    !************************************************
    ! Function    :     User interface message
    ! Programmer  :     Philippe Fleischmann
    ! Date        :     2019.02.22
    !***************** ETH Zurich *******************
    !
    FUNC string f_RRC_UIMsg(string stMsgHeader,string stMsgL1,\string stMsgL2,\string stMsgL3,\string stMsgL4,\string stMsgL5,string stBtn1\string stBtn2\string stBtn3\string stBtn4\string stBtn5,icondata icIcon)
        VAR num nAnswer;
        VAR string stMsg{5};
        VAR string stBtn{5};
        VAR string stAnswer;
        !
        ! Initialize variables
        stMsg:=["","","","",""];
        stBtn:=["","","","",""];
        !
        ! Load meassge
        stMsg{1}:=stMsgL1;
        IF Present(stMsgL2) stMsg{2}:=stMsgL2;
        IF Present(stMsgL3) stMsg{3}:=stMsgL3;
        IF Present(stMsgL4) stMsg{4}:=stMsgL4;
        IF Present(stMsgL5) stMsg{5}:=stMsgL5;
        !
        ! Load buttons
        stBtn{1}:=stBtn1;
        IF Present(stBtn2) stBtn{2}:=stBtn2;
        IF Present(stBtn3) stBtn{3}:=stBtn3;
        IF Present(stBtn4) stBtn{4}:=stBtn4;
        IF Present(stBtn5) stBtn{5}:=stBtn5;
        !
        ! Msg for user
        nAnswer:=UIMessageBox(
            \Header:=stMsgHeader
            \MsgArray:=stMsg
            \BtnArray:=stBtn
            \Icon:=icIcon);
        !
        ! handle user answer
        IF nAnswer=1 stAnswer:=stBtn{1};
        IF nAnswer=2 stAnswer:=stBtn{2};
        IF nAnswer=3 stAnswer:=stBtn{3};
        IF nAnswer=4 stAnswer:=stBtn{4};
        IF nAnswer=5 stAnswer:=stBtn{5};
        !
        ! Return user answer as string
        RETURN stAnswer;
    ERROR
        ! Placeholder for Error Code...
    ENDFUNC

    !************************************************
    ! Function    :     User interface numerical entry
    ! Programmer  :     Philippe Fleischmann
    ! Date        :     2019.02.22
    !***************** ETH Zurich *******************
    !
    FUNC num f_RRC_UINumEntry(string stMsgHeader,string stMsgL1,\string stMsgL2,\string stMsgL3,\string stMsgL4,\string stMsgL5,num nMin,num nMax,\num nDefault,icondata icIcon)
        VAR string stMsg{5};
        VAR num nAnswer;
        VAR num nInitValue;
        !
        ! Initialize variables
        stMsg:=["","","","",""];
        nInitValue:=nMin;
        !
        ! Load meassge
        stMsg{1}:=stMsgL1;
        IF Present(stMsgL2) stMsg{2}:=stMsgL2;
        IF Present(stMsgL3) stMsg{3}:=stMsgL3;
        IF Present(stMsgL4) stMsg{4}:=stMsgL4;
        IF Present(stMsgL5) stMsg{5}:=stMsgL5;
        !
        ! Use default value when present
        IF Present(nDefault) nInitValue:=nDefault;
        !
        ! Msg for user
        nAnswer:=Round(UINumEntry(
            \Header:=stMsgHeader
            \MsgArray:=stMsg
            \Icon:=icIcon
            \InitValue:=nInitValue
            \MinValue:=nMin
            \MaxValue:=nMax)\Dec:=1);
        !
        ! Return user answer as string
        RETURN nAnswer;
    ERROR
        ! Placeholder for Error Code...
    ENDFUNC


ENDMODULE

--- Backups/vIRB4600-40-2.55-RW11/RAPID/TASK2/SYSMOD/RRC_Base_Feedback_Ctrl.sys ---
MODULE RRC_Base_Feedback_Ctrl(SYSMODULE)
    !***********************************************************************************
    !
    ! ETH Zurich / Robotic Fabrication Lab
    ! HIB C 13 / Stefano-Franscini-Platz 1
    ! CH-8093 Zurich
    !
    !***********************************************************************************
    !
    ! PROJECT     :  RRC - Rapid Robot Communication
    !
    ! FUNCTION    :  Base Feedback Library
    !
    ! AUTHOR      :  Philippe Fleischmann
    !
    ! EMAIL       :  rrc@arch.ethz.ch
    !
    ! HISTORY     :  2019.02.22
    !
    ! Copyright   :  ETH Zurich (CH) 2019
    !                - Philippe Fleischmann
    !                - Michael Lyrenmann
    !                - Gonzalo Casas
    !
    ! License     :  This code base is governed by an EULA (End-User License Agreement)
    !                which you have received together with the software.
    !                You are not allowed to use the software on a real robots
    !                without a signed EULA.
    !
    !                A copy of the EULA content is in the controller task (T_CTRL).
    !
    !***********************************************************************************

    !************************************************
    ! Function    :     Feedback add string
    ! Programmer  :     Philippe Fleischmann
    ! Date        :     2019.02.22
    !***************** ETH Zurich *******************
    !
    PROC r_RRC_FAddString(string stString)
        !
        ! Increase feedback string counter
        Incr n_RRC_CounterFStr{n_RRC_ChaNr};
        !
        ! Select string to add
        TEST n_RRC_CounterFStr{n_RRC_ChaNr}
        CASE 1:
            !
            ! Add string
            bm_RRC_ActSenMsgCtrl{n_RRC_ChaNr}.Data.St1:=stString;
        CASE 2:
            !
            ! Add string
            bm_RRC_ActSenMsgCtrl{n_RRC_ChaNr}.Data.St2:=stString;
        CASE 3:
            !
            ! Add string
            bm_RRC_ActSenMsgCtrl{n_RRC_ChaNr}.Data.St3:=stString;
        CASE 4:
            !
            ! Add string
            bm_RRC_ActSenMsgCtrl{n_RRC_ChaNr}.Data.St4:=stString;
        CASE 5:
            !
            ! Add string
            bm_RRC_ActSenMsgCtrl{n_RRC_ChaNr}.Data.St5:=stString;
        DEFAULT:
            !
            ! Program error
            r_RRC_ProgError;
        ENDTEST
        !
        ! Update string counter
        bm_RRC_ActSenMsgCtrl{n_RRC_ChaNr}.Data.St_Cnt:=n_RRC_CounterFStr{n_RRC_ChaNr};
        RETURN ;
    ERROR
        ! Placeholder for Error Code...
    ENDPROC

    !************************************************
    ! Function    :     Feedback add value
    ! Programmer  :     Philippe Fleischmann
    ! Date        :     2019.02.22
    !***************** ETH Zurich *******************
    !
    PROC r_RRC_FAddValue(num nValue)
        !
        ! Increase feedback value counter
        Incr n_RRC_CounterFVal{n_RRC_ChaNr};
        !
        ! Select value to add
        TEST n_RRC_CounterFVal{n_RRC_ChaNr}
        CASE 1:
            !
            ! Add value
            bm_RRC_ActSenMsgCtrl{n_RRC_ChaNr}.Data.V1:=nValue;
        CASE 2:
            !
            ! Add value
            bm_RRC_ActSenMsgCtrl{n_RRC_ChaNr}.Data.V2:=nValue;
        CASE 3:
            !
            ! Add value
            bm_RRC_ActSenMsgCtrl{n_RRC_ChaNr}.Data.V3:=nValue;
        CASE 4:
            !
            ! Add value
            bm_RRC_ActSenMsgCtrl{n_RRC_ChaNr}.Data.V4:=nValue;
        CASE 5:
            !
            ! Add value
            bm_RRC_ActSenMsgCtrl{n_RRC_ChaNr}.Data.V5:=nValue;
        CASE 6:
            !
            ! Add value
            bm_RRC_ActSenMsgCtrl{n_RRC_ChaNr}.Data.V6:=nValue;
        CASE 7:
            !
            ! Add value
            bm_RRC_ActSenMsgCtrl{n_RRC_ChaNr}.Data.V7:=nValue;
        CASE 8:
            !
            ! Add value
            bm_RRC_ActSenMsgCtrl{n_RRC_ChaNr}.Data.V8:=nValue;
        CASE 9:
            !
            ! Add value
            bm_RRC_ActSenMsgCtrl{n_RRC_ChaNr}.Data.V9:=nValue;
        CASE 10:
            !
            ! Add value
            bm_RRC_ActSenMsgCtrl{n_RRC_ChaNr}.Data.V10:=nValue;
        CASE 11:
            !
            ! Add value
            bm_RRC_ActSenMsgCtrl{n_RRC_ChaNr}.Data.V11:=nValue;
        CASE 12:
            !
            ! Add value
            bm_RRC_ActSenMsgCtrl{n_RRC_ChaNr}.Data.V12:=nValue;
        CASE 13:
            !
            ! Add value
            bm_RRC_ActSenMsgCtrl{n_RRC_ChaNr}.Data.V13:=nValue;
        CASE 14:
            !
            ! Add value
            bm_RRC_ActSenMsgCtrl{n_RRC_ChaNr}.Data.V14:=nValue;
        CASE 15:
            !
            ! Add value
            bm_RRC_ActSenMsgCtrl{n_RRC_ChaNr}.Data.V15:=nValue;
        CASE 16:
            !
            ! Add value
            bm_RRC_ActSenMsgCtrl{n_RRC_ChaNr}.Data.V16:=nValue;
        CASE 17:
            !
            ! Add value
            bm_RRC_ActSenMsgCtrl{n_RRC_ChaNr}.Data.V17:=nValue;
        CASE 18:
            !
            ! Add value
            bm_RRC_ActSenMsgCtrl{n_RRC_ChaNr}.Data.V18:=nValue;
        CASE 19:
            !
            ! Add value
            bm_RRC_ActSenMsgCtrl{n_RRC_ChaNr}.Data.V19:=nValue;
        CASE 20:
            !
            ! Add value
            bm_RRC_ActSenMsgCtrl{n_RRC_ChaNr}.Data.V20:=nValue;
        CASE 21:
            !
            ! Add value
            bm_RRC_ActSenMsgCtrl{n_RRC_ChaNr}.Data.V21:=nValue;
        CASE 22:
            !
            ! Add value
            bm_RRC_ActSenMsgCtrl{n_RRC_ChaNr}.Data.V22:=nValue;
        CASE 23:
            !
            ! Add value
            bm_RRC_ActSenMsgCtrl{n_RRC_ChaNr}.Data.V23:=nValue;
        CASE 24:
            !
            ! Add value
            bm_RRC_ActSenMsgCtrl{n_RRC_ChaNr}.Data.V24:=nValue;
        CASE 25:
            !
            ! Add value
            bm_RRC_ActSenMsgCtrl{n_RRC_ChaNr}.Data.V25:=nValue;
        CASE 26:
            !
            ! Add value
            bm_RRC_ActSenMsgCtrl{n_RRC_ChaNr}.Data.V26:=nValue;
        CASE 27:
            !
            ! Add value
            bm_RRC_ActSenMsgCtrl{n_RRC_ChaNr}.Data.V27:=nValue;
        CASE 28:
            !
            ! Add value
            bm_RRC_ActSenMsgCtrl{n_RRC_ChaNr}.Data.V28:=nValue;
        CASE 29:
            !
            ! Add value
            bm_RRC_ActSenMsgCtrl{n_RRC_ChaNr}.Data.V29:=nValue;
        CASE 30:
            !
            ! Add value
            bm_RRC_ActSenMsgCtrl{n_RRC_ChaNr}.Data.V30:=nValue;
        DEFAULT:
            !
            ! Program error
            r_RRC_ProgError;
        ENDTEST
        !
        ! Update value counter
        bm_RRC_ActSenMsgCtrl{n_RRC_ChaNr}.Data.V_Cnt:=n_RRC_CounterFVal{n_RRC_ChaNr};
        RETURN ;
    ERROR
        ! Placeholder for Error Code...
    ENDPROC

    !************************************************
    ! Function    :     Feedback done
    ! Programmer  :     Philippe Fleischmann
    ! Date        :     2019.02.22
    !***************** ETH Zurich *******************
    !
    PROC r_RRC_FDone()
        !
        ! Add Sqz_ID from Client in Feedback ID
        bm_RRC_ActSenMsgCtrl{n_RRC_ChaNr}.Data.F_ID:=bm_RRC_RecBufferCtrl{n_RRC_ChaNr,n_RRC_ReadPtrRecBuf{n_RRC_ChaNr}}.Data.S_ID;
        !
        ! Instruction
        bm_RRC_ActSenMsgCtrl{n_RRC_ChaNr}.Data.Instr:=bm_RRC_RecBufferCtrl{n_RRC_ChaNr,n_RRC_ReadPtrRecBuf{n_RRC_ChaNr}}.Data.Instr;
        !
        ! Feedback
        bm_RRC_ActSenMsgCtrl{n_RRC_ChaNr}.Data.Feedb:="Controller Done";
        RETURN ;
    ERROR
        ! Placeholder for Error Code...
    ENDPROC

    !************************************************
    ! Function    :     Cycle Feedback done
    ! Programmer  :     Philippe Fleischmann
    ! Date        :     2019.02.22
    !***************** ETH Zurich *******************
    !
    PROC r_RRC_CyFDone()
        !
        ! Add cyclic jop Sqz_ID from cyclic job start instruction
        bm_RRC_ActSenMsgCtrl{n_RRC_ChaNr}.Data.F_ID:=n_RRC_CyJobStart_S_ID{n_RRC_ChaNr};
        !
        ! Add cyclic jop instruction
        bm_RRC_ActSenMsgCtrl{n_RRC_ChaNr}.Data.Instr:=st_RRC_CyclicJob{n_RRC_ChaNr};
        !
        ! Feedback
        bm_RRC_ActSenMsgCtrl{n_RRC_ChaNr}.Data.Feedb:="Controller Done";
        RETURN ;
    ERROR
        ! Placeholder for Error Code...
    ENDPROC

    !************************************************
    ! Function    :     Feedback error
    ! Programmer  :     Philippe Fleischmann
    ! Date        :     2019.02.22
    !***************** ETH Zurich *******************
    !
    PROC r_RRC_FError()
        !
        ! Feedback error with feedback code
        bm_RRC_ActSenMsgCtrl{n_RRC_ChaNr}.Data.Feedb:="Controller Done FError "+NumToStr(bm_RRC_RecBufferCtrl{n_RRC_ChaNr,n_RRC_ReadPtrRecBuf{n_RRC_ChaNr}}.Data.F_Lev,0);
        RETURN ;
    ERROR
        ! Placeholder for Error Code...
    ENDPROC
ENDMODULE

--- Backups/vIRB4600-40-2.55-RW11/RAPID/TASK2/SYSMOD/RRC_Base_Instructions_Ctrl.sys ---
MODULE RRC_Base_Instructions_Ctrl(SYSMODULE)
    !***********************************************************************************
    !
    ! ETH Zurich / Robotic Fabrication Lab
    ! HIB C 13 / Stefano-Franscini-Platz 1
    ! CH-8093 Zurich
    !
    !***********************************************************************************
    !
    ! PROJECT     :  RRC - Rapid Robot Communication
    !
    ! FUNCTION    :  Base Instracion Library for controller
    !
    ! AUTHOR      :  Philippe Fleischmann
    !
    ! EMAIL       :  rrc@arch.ethz.ch
    !
    ! HISTORY     :  2019.02.22
    !
    ! Copyright   :  ETH Zurich (CH) 2019
    !                - Philippe Fleischmann
    !                - Michael Lyrenmann
    !                - Gonzalo Casas
    !
    ! License     :  This code base is governed by an EULA (End-User License Agreement)
    !                which you have received together with the software.
    !                You are not allowed to use the software on a real robots
    !                without a signed EULA.
    !
    !                A copy of the EULA content is in the controller task (T_CTRL).
    !
    !***********************************************************************************

    !************************************************
    ! Function    :     Dummy
    ! Programmer  :     Philippe Fleischmann
    ! Date        :     2019.02.22
    !***************** ETH Zurich *******************
    !
    PROC r_RRC_Dummy()
        !
        ! Just a dummy procedure for communication tests
        !
        ! Read the current Sequnce ID
        n_RRC_Act_S_ID:=bm_RRC_RecBufferCtrl{n_RRC_ChaNr,n_RRC_ReadPtrRecBuf{n_RRC_ChaNr}}.Data.S_ID;
        !
        ! Feedback
        IF bm_RRC_RecBufferCtrl{n_RRC_ChaNr,n_RRC_ReadPtrRecBuf{n_RRC_ChaNr}}.Data.F_Lev>0 THEN
            !
            ! Cenerate feedback
            TEST bm_RRC_RecBufferCtrl{n_RRC_ChaNr,n_RRC_ReadPtrRecBuf{n_RRC_ChaNr}}.Data.F_Lev
            CASE 1:
                !nChaNr
                ! Instruction done
                r_RRC_FDone;
            DEFAULT:
                !
                ! Feedback not supported
                r_RRC_FError;
            ENDTEST
            !
            ! Move message in send buffer
            r_RRC_MovMsgToSenBufCtrl n_RRC_ChaNr;
        ENDIF
        RETURN ;
    ERROR
        ! Placeholder for Error Code...
    ENDPROC

    !************************************************
    ! Function    :     Read actual jointtarget
    ! Programmer  :     Philippe Fleischmann
    ! Date        :     2019.02.22
    !***************** ETH Zurich *******************
    !
    PROC r_RRC_GetJointT()
        !
        ! Read current joint position
        jp_RRC_Act:=CJointT(\TaskName:=st_RRC_ChaTask);
        !
        ! Add robot axis values to feedback
        r_RRC_FAddValue jp_RRC_Act.robax.rax_1;
        r_RRC_FAddValue jp_RRC_Act.robax.rax_2;
        r_RRC_FAddValue jp_RRC_Act.robax.rax_3;
        r_RRC_FAddValue jp_RRC_Act.robax.rax_4;
        r_RRC_FAddValue jp_RRC_Act.robax.rax_5;
        r_RRC_FAddValue jp_RRC_Act.robax.rax_6;
        !
        ! Add external axis values to feedback
        r_RRC_FAddValue jp_RRC_Act.extax.eax_a;
        r_RRC_FAddValue jp_RRC_Act.extax.eax_b;
        r_RRC_FAddValue jp_RRC_Act.extax.eax_c;
        r_RRC_FAddValue jp_RRC_Act.extax.eax_d;
        r_RRC_FAddValue jp_RRC_Act.extax.eax_e;
        r_RRC_FAddValue jp_RRC_Act.extax.eax_f;
        !
        ! Add cyclic feedback instruction done
        r_RRC_CyFDone;
        !
        ! Feedback
        IF bm_RRC_RecBufferCtrl{n_RRC_ChaNr,n_RRC_ReadPtrRecBuf{n_RRC_ChaNr}}.Data.F_Lev>1 THEN
            !
            ! Check additional feedback
            TEST bm_RRC_RecBufferCtrl{n_RRC_ChaNr,n_RRC_ReadPtrRecBuf{n_RRC_ChaNr}}.Data.F_Lev
            CASE 10001:
                !
                ! add robot position
                !* r_RRC_FPos bm_RRC_RecBufferRob{n_RRC_ChaNr,n_RRC_ReadPtrRecBuf}.Data.F_Lev;
            DEFAULT:
                !
                ! Not defined
                !
                ! Feedback not supported
                r_RRC_FError;
            ENDTEST
        ENDIF
        !
        ! Move message in send buffer
        r_RRC_MovMsgToSenBufCtrl n_RRC_ChaNr;
        RETURN ;
    ERROR
        ! Placeholder for Error Code...
    ENDPROC

    !************************************************
    ! Function    :     Get robtarget
    ! Programmer  :     Philippe Fleischmann
    ! Date        :     2019.02.22
    !***************** ETH Zurich *******************
    !
    PROC r_RRC_GetRobT()
        !
        ! Read current joint position
        p_RRC_Act:=CRobT(\TaskName:=st_RRC_ChaTask);
        !
        ! Add translastion values to feedback
        r_RRC_FAddValue p_RRC_Act.trans.x;
        r_RRC_FAddValue p_RRC_Act.trans.y;
        r_RRC_FAddValue p_RRC_Act.trans.z;
        !
        ! Add rotation values to feedback
        r_RRC_FAddValue p_RRC_Act.rot.q1;
        r_RRC_FAddValue p_RRC_Act.rot.q2;
        r_RRC_FAddValue p_RRC_Act.rot.q3;
        r_RRC_FAddValue p_RRC_Act.rot.q4;
        !
        ! Add external axis values to feedback
        r_RRC_FAddValue p_RRC_Act.extax.eax_a;
        r_RRC_FAddValue p_RRC_Act.extax.eax_b;
        r_RRC_FAddValue p_RRC_Act.extax.eax_c;
        r_RRC_FAddValue p_RRC_Act.extax.eax_d;
        r_RRC_FAddValue p_RRC_Act.extax.eax_e;
        r_RRC_FAddValue p_RRC_Act.extax.eax_f;
        !
        ! Add standard feedback instruction done
        r_RRC_FDone;
        !
        ! Feedback
        IF bm_RRC_RecBufferCtrl{n_RRC_ChaNr,n_RRC_ReadPtrRecBuf{n_RRC_ChaNr}}.Data.F_Lev>1 THEN
            !
            ! Check additional feedback
            TEST bm_RRC_RecBufferCtrl{n_RRC_ChaNr,n_RRC_ReadPtrRecBuf{n_RRC_ChaNr}}.Data.F_Lev
            CASE 10001:
                !
                ! add robot position
                !* r_RRC_FPos bm_RRC_RecBufferRob{n_RRC_ChaNr,n_RRC_ReadPtrRecBuf}.Data.F_Lev;
            DEFAULT:
                !
                ! Not defined
                !
                ! Feedback not supported
                r_RRC_FError;
            ENDTEST
        ENDIF
        !
        ! Move message in send buffer
        r_RRC_MovMsgToSenBufCtrl n_RRC_ChaNr;
        RETURN ;
    ERROR
        ! Placeholder for Error Code...
    ENDPROC

    !************************************************
    ! Function    :     Stop
    ! Programmer  :     Philippe Fleischmann
    ! Date        :     2019.02.22
    !***************** ETH Zurich *******************
    !
    PROC r_RRC_Stop()
        !
        ! Stop task
        Stop;
        !
        ! Feedback
        IF bm_RRC_RecBufferCtrl{n_RRC_ChaNr,n_RRC_ReadPtrRecBuf{n_RRC_ChaNr}}.Data.F_Lev>0 THEN
            !
            ! Cenerate feedback
            TEST bm_RRC_RecBufferCtrl{n_RRC_ChaNr,n_RRC_ReadPtrRecBuf{n_RRC_ChaNr}}.Data.F_Lev
            CASE 1:
                !
                ! Instruction done
                r_RRC_FDone;
            DEFAULT:
                !
                ! Feedback not supported
                r_RRC_FError;
            ENDTEST
            !
            ! Move message in send buffer
            r_RRC_MovMsgToSenBufCtrl n_RRC_ChaNr;
        ENDIF
        RETURN ;
    ERROR
        ! Placeholder for Error Code...
    ENDPROC

    !************************************************
    ! Function    :     Teachpendant Write
    ! Programmer  :     Philippe Fleischmann
    ! Date        :     2019.02.22
    !***************** ETH Zurich *******************
    !
    PROC r_RRC_TPWrite()
        !
        ! Read acceleration
        st_RRC_TPWrite{n_RRC_ChaNr}:=bm_RRC_RecBufferCtrl{n_RRC_ChaNr,n_RRC_ReadPtrRecBuf{n_RRC_ChaNr}}.Data.St1;
        !
        ! Clear panel
        TPErase;
        !
        ! Show message to user
        TPWrite st_RRC_TPWrite{n_RRC_ChaNr};
        !
        ! Feedback
        IF bm_RRC_RecBufferCtrl{n_RRC_ChaNr,n_RRC_ReadPtrRecBuf{n_RRC_ChaNr}}.Data.F_Lev>0 THEN
            !
            ! Cenerate feedback
            TEST bm_RRC_RecBufferCtrl{n_RRC_ChaNr,n_RRC_ReadPtrRecBuf{n_RRC_ChaNr}}.Data.F_Lev
            CASE 1:
                !
                ! Instruction done
                r_RRC_FDone;
            DEFAULT:
                !
                ! Feedback not supported
                r_RRC_FError;
            ENDTEST
            !
            ! Move message in send buffer
            r_RRC_MovMsgToSenBufCtrl n_RRC_ChaNr;
        ENDIF
        RETURN ;
    ERROR
        ! Placeholder for Error Code...
    ENDPROC

    !************************************************
    ! Function    :     Cyclic job start
    ! Programmer  :     Philippe Fleischmann
    ! Date        :     2019.02.22
    !***************** ETH Zurich *******************
    !
    PROC r_RRC_CyJobStart()
        !
        ! Read cyclic jop Sqz_ID
        n_RRC_CyJobStart_S_ID{n_RRC_ChaNr}:=bm_RRC_RecBufferCtrl{n_RRC_ChaNr,n_RRC_ReadPtrRecBuf{n_RRC_ChaNr}}.Data.S_ID;
        !
        ! Read cyclic job
        st_RRC_CyclicJob{n_RRC_ChaNr}:=bm_RRC_RecBufferCtrl{n_RRC_ChaNr,n_RRC_ReadPtrRecBuf{n_RRC_ChaNr}}.Data.St1;
        !
        ! Read cycle minimal time
        n_RRC_MinCycleTime{n_RRC_ChaNr}:=bm_RRC_RecBufferCtrl{n_RRC_ChaNr,n_RRC_ReadPtrRecBuf{n_RRC_ChaNr}}.Data.V1;
        !
        ! Activate cyclic job
        b_RRC_CyclicJob{n_RRC_ChaNr}:=TRUE;
        !
        ! Start cycle clock
        ClkStart ck_RRC_CycleJob{n_RRC_ChaNr};
        !
        ! Feedback
        IF bm_RRC_RecBufferCtrl{n_RRC_ChaNr,n_RRC_ReadPtrRecBuf{n_RRC_ChaNr}}.Data.F_Lev>0 THEN
            !
            ! Cenerate feedback
            TEST bm_RRC_RecBufferCtrl{n_RRC_ChaNr,n_RRC_ReadPtrRecBuf{n_RRC_ChaNr}}.Data.F_Lev
            CASE 1:
                !nChaNr
                ! Instruction done
                r_RRC_FDone;
            DEFAULT:
                !
                ! Feedback not supported
                r_RRC_FError;
            ENDTEST
            !
            ! Move message in send buffer
            r_RRC_MovMsgToSenBufCtrl n_RRC_ChaNr;
        ENDIF
        !
        ! Event log message
        r_RRC_EvLogMsg st_RRC_EvLogMsgHeader,"Cyclic job channel "+NumToStr(n_RRC_ChaNr,0)+" started with job: "+st_RRC_CyclicJob{n_RRC_ChaNr};
        RETURN ;
    ERROR
        ! Placeholder for Error Code...
    ENDPROC

    !************************************************
    ! Function    :     Cyclic job end
    ! Programmer  :     Philippe Fleischmann
    ! Date        :     2019.02.22
    !***************** ETH Zurich *******************
    !
    PROC r_RRC_CyJobEnd()
        !
        ! Stop and reset cycle clock
        ClkStop ck_RRC_CycleJob{n_RRC_ChaNr};
        ClkReset ck_RRC_CycleJob{n_RRC_ChaNr};
        !
        ! Deactivate cyclic job
        b_RRC_CyclicJob{n_RRC_ChaNr}:=FALSE;
        !
        ! Feedback
        IF bm_RRC_RecBufferCtrl{n_RRC_ChaNr,n_RRC_ReadPtrRecBuf{n_RRC_ChaNr}}.Data.F_Lev>0 THEN
            !
            ! Cenerate feedback
            TEST bm_RRC_RecBufferCtrl{n_RRC_ChaNr,n_RRC_ReadPtrRecBuf{n_RRC_ChaNr}}.Data.F_Lev
            CASE 1:
                !nChaNr
                ! Instruction done
                r_RRC_FDone;
            DEFAULT:
                !
                ! Feedback not supported
                r_RRC_FError;
            ENDTEST
            !
            ! Move message in send buffer
            r_RRC_MovMsgToSenBufCtrl n_RRC_ChaNr;
        ENDIF
        !
        ! Event log message
        r_RRC_EvLogMsg st_RRC_EvLogMsgHeader,"Cyclic job channel "+NumToStr(n_RRC_ChaNr,0)+" ended with job: "+st_RRC_CyclicJob{n_RRC_ChaNr};
        RETURN ;
    ERROR
        ! Placeholder for Error Code...
    ENDPROC

    !************************************************
    ! Function    :     Cyclic job test
    ! Programmer  :     Philippe Fleischmann
    ! Date        :     2019.02.22
    !***************** ETH Zurich *******************
    !
    PROC r_RRC_CyJobTest()
        !
        ! Increase cycle time
        Incr n_RRC_ActCycle{n_RRC_ChaNr};
        !
        ! Write cycle number and ccurrent cycle time
        TPWrite "Cycle Nr: "+NumToStr(n_RRC_ActCycle{n_RRC_ChaNr},0)+" Cycle Time: "+NumToStr(n_RRC_LastCycleTime{n_RRC_ChaNr},3);
        !
        ! Feedback
        IF bm_RRC_RecBufferCtrl{n_RRC_ChaNr,n_RRC_ReadPtrRecBuf{n_RRC_ChaNr}}.Data.F_Lev>0 THEN
            !
            ! Cenerate feedback
            TEST bm_RRC_RecBufferCtrl{n_RRC_ChaNr,n_RRC_ReadPtrRecBuf{n_RRC_ChaNr}}.Data.F_Lev
            CASE 1:
                !nChaNr
                ! Instruction done
                r_RRC_FDone;
            DEFAULT:
                !
                ! Feedback not supported
                r_RRC_FError;
            ENDTEST
            !
            ! Move message in send buffer
            r_RRC_MovMsgToSenBufCtrl n_RRC_ChaNr;
        ENDIF
        !
        ! Event log message
        r_RRC_EvLogMsg st_RRC_EvLogMsgHeader,"Cyclic job channel "+NumToStr(n_RRC_ChaNr,0)+" running with job: "+st_RRC_CyclicJob{n_RRC_ChaNr};
        RETURN ;
    ERROR
        ! Placeholder for Error Code...
    ENDPROC
ENDMODULE

--- Backups/vIRB4600-40-2.55-RW11/RAPID/TASK2/SYSMOD/RRC_Config_Ctrl.sys ---
MODULE RRC_Config_Ctrl(SYSMODULE)
    !***********************************************************************************
    !
    ! ETH Zurich / Robotic Fabrication Lab
    ! HIB C 13 / Stefano-Franscini-Platz 1
    ! CH-8093 Zurich
    !
    !***********************************************************************************
    !
    ! PROJECT     :  RRC - Rapid Robot Communication
    !
    ! FUNCTION    :  Configuration modul for the project
    !
    ! AUTHOR      :  Philippe Fleischmann
    !
    ! EMAIL       :  rrc@arch.ethz.ch
    !
    ! HISTORY     :  2019.02.22
    !
    ! Copyright   :  ETH Zurich (CH) 2019
    !                - Philippe Fleischmann
    !                - Michael Lyrenmann
    !                - Gonzalo Casas
    !
    ! License     :  This code base is governed by an EULA (End-User License Agreement)
    !                which you have received together with the software.
    !                You are not allowed to use the software on a real robots
    !                without a signed EULA.
    !
    !                A copy of the EULA content is in the controller task (T_CTRL).
    !
    !***********************************************************************************

    !************************************************
    ! Function    :     Initialize Cell
    ! Programmer  :     Philippe Fleischmann
    ! Date        :     2019.02.22
    !***************** ETH Zurich *******************
    !
    PROC r_RRC_RRC_Config()
        !
        ! Current controller job, used from the RFL Controller project selection (st_RFL_CurCtrlJob)
        ! Default value "RRC"
        st_RRC_CurCtrlJob:="RRC";
        !
        ! Tasklists
        tl_RRC_All:=[["T_CTRL"],["T_RX"],["T_TX"],["T_ROB1"],[""],[""],[""]];
        !
        ! Channel 1
        ch_RRC_Channels.Ch_1.T_Name:="T_ROB1";
        ch_RRC_Channels.Ch_1.Ch_Nr:=1;
        !
        ! Channel 2
        ch_RRC_Channels.Ch_2.T_Name:="T_ROB2";
        ch_RRC_Channels.Ch_2.Ch_Nr:=2;
        !
        ! Channel 3
        ch_RRC_Channels.Ch_3.T_Name:="T_ROB3";
        ch_RRC_Channels.Ch_3.Ch_Nr:=3;
        !
        ! Channel 4
        ch_RRC_Channels.Ch_4.T_Name:="T_ROB4";
        ch_RRC_Channels.Ch_4.Ch_Nr:=4;
        !
        ! IP Address
        b_RRC_AutoIPAddress:=TRUE;
        st_RRC_IP_AddressMan:="192.168.125.1";
        !
        ! Ports
        b_RRC_VirtualCustomPorts:=FALSE;
        n_RRC_ViCustomSocketPortRec:=[31101,31102,31103,31104];
        n_RRC_ViCustomSocketPortSen:=[31201,31202,31203,31204];
        !
        ! Roboter 1
        b_RRC_Com{n_RRC_R1_ChaNr}:=TRUE;
        b_RRC_SIDCheck{n_RRC_R1_ChaNr}:=TRUE;
        b_RRC_SIDErrorStop{n_RRC_R1_ChaNr}:=FALSE;
        b_RRC_LogPro{n_RRC_R1_ChaNr}:=FALSE;
        !
        ! Roboter 2
        b_RRC_Com{n_RRC_R2_ChaNr}:=FALSE;
        b_RRC_SIDCheck{n_RRC_R2_ChaNr}:=FALSE;
        b_RRC_SIDErrorStop{n_RRC_R2_ChaNr}:=FALSE;
        b_RRC_LogPro{n_RRC_R2_ChaNr}:=FALSE;
        !
        ! Roboter 3
        b_RRC_Com{n_RRC_R3_ChaNr}:=FALSE;
        b_RRC_SIDCheck{n_RRC_R3_ChaNr}:=FALSE;
        b_RRC_SIDErrorStop{n_RRC_R3_ChaNr}:=FALSE;
        b_RRC_LogPro{n_RRC_R3_ChaNr}:=FALSE;
        !
        ! Roboter 4
        b_RRC_Com{n_RRC_R4_ChaNr}:=FALSE;
        b_RRC_SIDCheck{n_RRC_R4_ChaNr}:=FALSE;
        b_RRC_SIDErrorStop{n_RRC_R4_ChaNr}:=FALSE;
        b_RRC_LogPro{n_RRC_R4_ChaNr}:=FALSE;
        RETURN ;
    ERROR
        ! Placeholder for Error Code...
    ENDPROC

ENDMODULE

--- Backups/vIRB4600-40-2.55-RW11/RAPID/TASK2/SYSMOD/RRC_Control_Ctrl.sys ---
MODULE RRC_Control_Ctrl(SYSMODULE)
    !***********************************************************************************
    !
    ! ETH Zurich / Robotic Fabrication Lab
    ! HIB C 13 / Stefano-Franscini-Platz 1
    ! CH-8093 Zurich
    !
    !***********************************************************************************
    !
    ! PROJECT     :  RRC - Rapid Robot Communication
    !
    ! FUNCTION    :  Control modul for the project
    !
    ! AUTHOR      :  Philippe Fleischmann
    !
    ! EMAIL       :  rrc@arch.ethz.ch
    !
    ! HISTORY     :  2019.02.22
    !
    ! Copyright   :  ETH Zurich (CH) 2019
    !                - Philippe Fleischmann
    !                - Michael Lyrenmann
    !                - Gonzalo Casas
    !
    ! License     :  This code base is governed by an EULA (End-User License Agreement)
    !                which you have received together with the software.
    !                You are not allowed to use the software on a real robots
    !                without a signed EULA.
    !
    !                A copy of the EULA content is in the controller task (T_CTRL).
    !
    !***********************************************************************************

    !************************************************
    ! Function    :     Main for Project RRC
    ! Programmer  :     Philippe Fleischmann
    ! Date        :     2019.02.22
    !***************** ETH Zurich *******************
    !
    PROC r_RRC_Main()
        !
        ! Configure communication
        %"r_"+st_RRC_CurCtrlJob+"_RRC_Config"%;
        !
        ! Clear Display
        TPErase;
        !
        ! Task synchronisation
        WaitSyncTask id_RRC_MainSta,tl_RRC_All;
        !
        ! Message for Operator
        TPWrite "RRC Main";
        !
        ! Init Project
        r_RRC_InitCell;
        !
        ! Production loop
        WHILE b_RRC_Run=TRUE DO
            !
            ! Check for single and cycle job
            IF b_RRC_Com{n_RRC_R1_ChaNr} r_RRC_CheckCtrlJob n_RRC_R1_ChaNr;
            !
            ! Check for single and cycle job
            IF b_RRC_Com{n_RRC_R2_ChaNr} r_RRC_CheckCtrlJob n_RRC_R2_ChaNr;
            !
            ! Check for single and cycle job
            IF b_RRC_Com{n_RRC_R3_ChaNr} r_RRC_CheckCtrlJob n_RRC_R3_ChaNr;
            !
            ! Check for single and cycle job
            IF b_RRC_Com{n_RRC_R4_ChaNr} r_RRC_CheckCtrlJob n_RRC_R4_ChaNr;
        ENDWHILE
        !
        ! Message for Operator
        TPWrite "RRC End";
        !
        ! Task synchronisation
        WaitSyncTask id_RRC_MainEnd,tl_RRC_All;
        !
        RETURN ;
    ERROR
        ! Placeholder for Error Code...
    ENDPROC

    !************************************************
    ! Function    :     Initialize Cell
    ! Programmer  :     Philippe Fleischmann
    ! Date        :     2019.02.22
    !***************** ETH Zurich *******************
    !
    PROC r_RRC_InitCell()
        !
        ! Initialize Global Variables
        r_RRC_InitGlobalVar;
        !
        ! Task synchronisation
        WaitSyncTask id_RRC_InitSta,tl_RRC_All;
        !
        ! Read system data
        r_RRC_ReadSysData;
        !
        ! Initialize IP Address
        r_RRC_InitIP;
        !
        ! Initialize Ports
        r_RRC_InitPorts;
        !
        ! Initialize Variables
        r_RRC_InitVar;
        !
        ! Task synchronisation controller data done
        WaitSyncTask id_RRC_InitCtrl,tl_RRC_All;
        !
        ! Task synchronisation
        WaitSyncTask id_RRC_InitEnd,tl_RRC_All;
        !
        ! Check rrc connection and bring user message
        IF b_RRC_TaskReceiverOn=TRUE AND b_RRC_TaskSenderOn=TRUE THEN
            !
            ! User Message
            r_RRC_TPMsg " RRC-Connected ";
        ELSEIF b_RRC_TaskReceiverOn=TRUE AND b_RRC_TaskSenderOn=FALSE THEN
            !
            ! User Message
            r_RRC_TPMsg " RRC - Only receiver connected";

        ELSEIF b_RRC_TaskReceiverOn=FALSE AND b_RRC_TaskSenderOn=TRUE THEN
            !
            ! User Message
            r_RRC_TPMsg " RRC - Only sender connected";
        ELSE
            !
            ! User Message
            r_RRC_TPMsg " RRC - Not connected";
        ENDIF
        RETURN ;
    ERROR
        !
        ! Check error code
        TPWrite ""\Num:=ERRNO;
        TRYNEXT;
    ENDPROC

    !************************************************
    ! Function    :     Initialize global variables
    ! Programmer  :     Philippe Fleischmann
    ! Date        :     2019.02.22
    !***************** ETH Zurich *******************
    !
    PROC r_RRC_InitGlobalVar()
        !
        ! Reset task variables
        b_RRC_TaskReceiverOn:=FALSE;
        b_RRC_TaskSenderOn:=FALSE;
        RETURN ;
    ERROR
        ! Placeholder for Error Code...
    ENDPROC

    !************************************************
    ! Function    :     Initialize Variables
    ! Programmer  :     Philippe Fleischmann
    ! Date        :     2019.02.22
    !***************** ETH Zurich *******************
    !
    PROC r_RRC_InitVar()
        !
        ! Reset flag cycle job
        b_RRC_CyclicJob{n_RRC_R1_ChaNr}:=FALSE;
        b_RRC_CyclicJob{n_RRC_R2_ChaNr}:=FALSE;
        b_RRC_CyclicJob{n_RRC_R3_ChaNr}:=FALSE;
        b_RRC_CyclicJob{n_RRC_R4_ChaNr}:=FALSE;
        !
        ! Reset flag cycle time running
        b_RRC_CycleTimeRunnig{n_RRC_R1_ChaNr}:=FALSE;
        b_RRC_CycleTimeRunnig{n_RRC_R2_ChaNr}:=FALSE;
        b_RRC_CycleTimeRunnig{n_RRC_R3_ChaNr}:=FALSE;
        b_RRC_CycleTimeRunnig{n_RRC_R4_ChaNr}:=FALSE;
        !
        ! Reset Read pointer
        n_RRC_ReadPtrRecBuf{n_RRC_R1_ChaNr}:=1;
        n_RRC_ReadPtrRecBuf{n_RRC_R2_ChaNr}:=1;
        n_RRC_ReadPtrRecBuf{n_RRC_R3_ChaNr}:=1;
        n_RRC_ReadPtrRecBuf{n_RRC_R4_ChaNr}:=1;
        !
        ! Reset Counter Feedback Value
        n_RRC_CounterFStr{n_RRC_R1_ChaNr}:=0;
        n_RRC_CounterFStr{n_RRC_R2_ChaNr}:=0;
        n_RRC_CounterFStr{n_RRC_R3_ChaNr}:=0;
        n_RRC_CounterFStr{n_RRC_R4_ChaNr}:=0;
        !
        ! Reset Counter Feedback Value
        n_RRC_CounterFVal{n_RRC_R1_ChaNr}:=0;
        n_RRC_CounterFVal{n_RRC_R2_ChaNr}:=0;
        n_RRC_CounterFVal{n_RRC_R3_ChaNr}:=0;
        n_RRC_CounterFVal{n_RRC_R4_ChaNr}:=0;
        !
        ! Clear actual sending message
        bm_RRC_ActSenMsgCtrl{n_RRC_R1_ChaNr}:=bm_RRC_Empty;
        bm_RRC_ActSenMsgCtrl{n_RRC_R2_ChaNr}:=bm_RRC_Empty;
        bm_RRC_ActSenMsgCtrl{n_RRC_R3_ChaNr}:=bm_RRC_Empty;
        bm_RRC_ActSenMsgCtrl{n_RRC_R4_ChaNr}:=bm_RRC_Empty;
        !
        ! Placeholder
        RETURN ;
    ERROR
        ! Placeholder for Error Code...
    ENDPROC

    !************************************************
    ! Function    :     Initialize IP Addresse
    ! Programmer  :     Philippe Fleischmann
    ! Date        :     2019.02.22
    !***************** ETH Zurich *******************
    !
    PROC r_RRC_InitIP()
        !
        ! Check for automatic or manual IP Address
        IF b_RRC_AutoIPAddress=TRUE THEN
            !
            ! Automatic IP Address
            !
            ! Check for real or virtual controller
            IF RobOS()=TRUE THEN
                !
                ! Real controller
                !
                ! Read current IP Address
                st_RRC_IP_Address:=GetSysInfo(\LanIp);
            ELSE
                !
                ! Virtual controller
                !
                ! Set virtual IP Addresse
                st_RRC_IP_Address:=st_RRC_IP_AddressVC;
            ENDIF
        ELSE
            !
            ! Manual IP Address
            !
            ! Set manual IP Address
            st_RRC_IP_Address:=st_RRC_IP_AddressMan;
        ENDIF
        !
        ! Writ event log message for RobotStudio Output
        r_RRC_EvLogMsg st_RRC_EvLogMsgHeader,"Actual IP Address: "+st_RRC_IP_Address;
        RETURN ;
    ERROR
        ! Placeholder for Error Code...
    ENDPROC

    !************************************************
    ! Function    :     Initialize Ports
    ! Programmer  :     Philippe Fleischmann
    ! Date        :     2019.02.22
    !***************** ETH Zurich *******************
    !
    PROC r_RRC_InitPorts()
        !
        ! Default ports
        n_RRC_SocketPortRec:=n_RRC_DefaultSocketPortRec;
        n_RRC_SocketPortSen:=n_RRC_DefaultSocketPortSen;
        !
        ! Check for virtual custom ports
        IF RobOS()=FALSE AND b_RRC_VirtualCustomPorts=TRUE THEN
            !
            ! Set virtual custom ports
            n_RRC_SocketPortRec:=n_RRC_ViCustomSocketPortRec;
            n_RRC_SocketPortSen:=n_RRC_ViCustomSocketPortSen;
        ENDIF
        !
        ! Writ event log message for RobotStudio Output
        r_RRC_EvLogMsg st_RRC_EvLogMsgHeader,"Actual receiver ports: ["+NumToStr(n_RRC_SocketPortRec{1},0)+"; "+NumToStr(n_RRC_SocketPortRec{2},0)+"; "+NumToStr(n_RRC_SocketPortRec{3},0)+"; "+NumToStr(n_RRC_SocketPortRec{4},0)+"]";
        r_RRC_EvLogMsg st_RRC_EvLogMsgHeader,"Actual sender ports: ["+NumToStr(n_RRC_SocketPortSen{1},0)+"; "+NumToStr(n_RRC_SocketPortSen{2},0)+"; "+NumToStr(n_RRC_SocketPortSen{3},0)+"; "+NumToStr(n_RRC_SocketPortSen{4},0)+"]";
        RETURN ;
    ERROR
        ! Placeholder for Error Code...
    ENDPROC

    !************************************************
    ! Function    :     Read System Data
    ! Programmer  :     Philippe Fleischmann
    ! Date        :     2019.02.22
    !***************** ETH Zurich *******************
    !
    PROC r_RRC_ReadSysData()
        !
        ! Serial  number
        st_RRC_SerialNr:=GetSysInfo(\SerialNo);
        !
        ! Software version
        st_RRC_SoftwareVersion:=GetSysInfo(\SWVersion);
        !
        ! Software version name
        st_RRC_RobotWare:=GetSysInfo(\SWVersionName);
        !
        ! Controller ID
        st_RRC_ControllerID:=GetSysInfo(\CtrlId);
        !
        ! WAN IP address
        st_RRC_WAN_IP:=GetSysInfo(\LanIp);
        !
        ! Controller language
        st_RRC_ControllerLang:=GetSysInfo(\CtrlLang);
        !
        ! Active system
        st_RRC_SystemName:=GetSysInfo(\SystemName);
        RETURN ;
    ERROR
        ! Placeholder for Error Code...
    ENDPROC

    !************************************************
    ! Function    :     Check for controller job
    ! Programmer  :     Philippe Fleischmann
    ! Date        :     2019.02.22
    !***************** ETH Zurich *******************
    !
    PROC r_RRC_CheckCtrlJob(num nChaNr)
        !
        ! Write current channel number for the instructions
        n_RRC_ChaNr:=nChaNr;
        !
        ! Write current channel task name for the instructions
        TEST n_RRC_ChaNr
        CASE 1:
            !
            ! Set actual channel name
            st_RRC_ChaTask:=ch_RRC_Channels.Ch_1.T_Name;
        CASE 2:
            !
            ! Set actual channel name
            st_RRC_ChaTask:=ch_RRC_Channels.Ch_2.T_Name;
        CASE 3:
            !
            ! Set actual channel name
            st_RRC_ChaTask:=ch_RRC_Channels.Ch_3.T_Name;
        CASE 4:
            !
            ! Set actual channel name
            st_RRC_ChaTask:=ch_RRC_Channels.Ch_4.T_Name;
        DEFAULT:
        ENDTEST
        !
        ! Check for job in receiver buffer
        IF bm_RRC_RecBufferCtrl{n_RRC_ChaNr,n_RRC_ReadPtrRecBuf{n_RRC_ChaNr}}.startbit=TRUE THEN
            !
            ! Execute job from receiver buffer
            r_RRC_ExeJobFrmRecBuf;
            !
        ENDIF
        !
        ! Check cyclic job
        IF b_RRC_CyclicJob{n_RRC_ChaNr}=TRUE THEN
            !
            ! Check cycle time
            IF f_RRC_CyTiExpired()=TRUE THEN
                !
                ! Call cycle job
                %st_RRC_CyclicJob{n_RRC_ChaNr}%;
            ENDIF
        ENDIF
    ERROR
        ! Placeholder for Error Code...
    ENDPROC

    !************************************************
    ! Function    :     Execute job from reveicer buffer
    ! Programmer  :     Philippe Fleischmann
    ! Date        :     2019.02.22
    !***************** ETH Zurich *******************
    !
    PROC r_RRC_ExeJobFrmRecBuf()
        !
        ! Call instruction
        %bm_RRC_RecBufferCtrl{n_RRC_ChaNr,n_RRC_ReadPtrRecBuf{n_RRC_ChaNr}}.Data.Instr %;
        !
        ! Set job done
        bm_RRC_RecBufferCtrl{n_RRC_ChaNr,n_RRC_ReadPtrRecBuf{n_RRC_ChaNr}}.startbit:=FALSE;
        !
        ! Count read pointer
        IF n_RRC_ReadPtrRecBuf{n_RRC_ChaNr}<DIM(bm_RRC_RecBufferCtrl,2) THEN
            !
            ! Increas write pointer form buffer
            Incr n_RRC_ReadPtrRecBuf{n_RRC_ChaNr};
        ELSE
            !
            ! Restart with one
            n_RRC_ReadPtrRecBuf{n_RRC_ChaNr}:=1;
        ENDIF
        RETURN ;
    ERROR
        ! Placeholder for Error Code...
    ENDPROC

    !************************************************
    ! Function    :     Move message to send buffer controller
    ! Programmer  :     Philippe Fleischmann
    ! Date        :     2019.02.22
    !***************** ETH Zurich *******************
    !
    PROC r_RRC_MovMsgToSenBufCtrl(num nChaNr)
        !
        ! Count buffer pointer
        IF n_RRC_WritePtrSenBufCtrl{nChaNr}<DIM(bm_RRC_SenBufferCtrl,2) THEN
            !
            ! Increas write pointer form buffer
            Incr n_RRC_WritePtrSenBufCtrl{nChaNr};
        ELSE
            !
            ! Restart with one
            n_RRC_WritePtrSenBufCtrl{nChaNr}:=1;
        ENDIF
        !
        ! Check for bufferline free to write
        IF NOT bm_RRC_SenBufferCtrl{nChaNr,n_RRC_WritePtrSenBufCtrl{nChaNr}}.startbit=FALSE THEN
            !
            ! Wait for bufferline free to write
            WaitUntil bm_RRC_SenBufferCtrl{nChaNr,n_RRC_WritePtrSenBufCtrl{nChaNr}}.startbit=FALSE\PollRate:=0.004\Visualize\Header:="RRC MovMsgToSenBufMa"\Message:="Buffer full"\Icon:=iconInfo;
        ENDIF
        !
        ! Write data in buffer
        bm_RRC_SenBufferCtrl{nChaNr,n_RRC_WritePtrSenBufCtrl{nChaNr}}.Data:=bm_RRC_ActSenMsgCtrl{nChaNr}.Data;
        !
        ! Set Startbit
        bm_RRC_SenBufferCtrl{nChaNr,n_RRC_WritePtrSenBufCtrl{nChaNr}}.startbit:=TRUE;
        !
        ! Clear actual sending message
        bm_RRC_ActSenMsgCtrl{nChaNr}:=bm_RRC_Empty;
        !
        ! Reset Counter Feedback String and Value
        n_RRC_CounterFStr{nChaNr}:=0;
        n_RRC_CounterFVal{nChaNr}:=0;
        RETURN ;
    ERROR
        ! Placeholder for Error Code...
    ENDPROC

    !************************************************
    ! Function    :     Cycle time expired
    ! Programmer  :     Philippe Fleischmann
    ! Date        :     2019.02.22
    !***************** ETH Zurich *******************
    !
    FUNC bool f_RRC_CyTiExpired()
        !
        ! Read current cycle time
        n_RRC_ActCycleTime{n_RRC_ChaNr}:=ClkRead(ck_RRC_CycleJob{n_RRC_ChaNr});
        !
        ! Check cycle time expired
        IF n_RRC_ActCycleTime{n_RRC_ChaNr}>n_RRC_MinCycleTime{n_RRC_ChaNr} THEN
            !
            ! Store last cycle time
            n_RRC_LastCycleTime{n_RRC_ChaNr}:=n_RRC_ActCycleTime{n_RRC_ChaNr};
            !
            ! Reset clock
            ClkReset ck_RRC_CycleJob{n_RRC_ChaNr};
            ClkStart ck_RRC_CycleJob{n_RRC_ChaNr};
            !
            ! Cycle time expired
            RETURN TRUE;
        ELSE
            !
            ! Cycle time not expired
            RETURN FALSE;
        ENDIF
    ERROR
        ! Placeholder for Error Code...
    ENDFUNC


    !************************************************
    ! Function    :     ProgError
    ! Programmer  :     Philippe Fleischmann
    ! Date        :     2019.02.22
    !***************** ETH Zurich *******************
    !
    PROC r_RRC_ProgError()
        !
        ! User Info
        TPWrite "Program Error";
        !
        ! Stop Program
        Stop;
        RETURN ;
    ERROR
        ! Placeholder for Error Code...
    ENDPROC

ENDMODULE

--- Backups/vIRB4600-40-2.55-RW11/RAPID/TASK2/SYSMOD/RRC_DataGlobal_Ctrl.sys ---
MODULE RRC_DataGlobal_Ctrl(SYSMODULE)
    !***********************************************************************************
    !
    ! ETH Zurich / Robotic Fabrication Lab
    ! HIB C13 / Stefano-Franscini-Platz 1
    ! CH-8093 Zurich
    !
    !***********************************************************************************
    !
    ! PROJECT     :  RRC - Rapid Robot Communication
    !
    ! FUNCTION    :  Inclouds all project spezific global datas
    !
    ! AUTHOR      :  Philippe Fleischmann
    !
    ! EMAIL       :  rrc@arch.ethz.ch
    !
    ! HISTORY     :  2019.02.22
    !
    ! Copyright   :  ETH Zurich (CH) 2019
    !                - Philippe Fleischmann
    !                - Michael Lyrenmann
    !                - Gonzalo Casas
    !
    ! License     :  This code base is governed by an EULA (End-User License Agreement)
    !                which you have received together with the software.
    !                You are not allowed to use the software on a real robots
    !                without a signed EULA.
    !
    !                A copy of the EULA content is in the controller task (T_CTRL).
    !
    !***********************************************************************************

    !************************************************
    ! Declaration :     bool
    !************************************************
    !
    PERS bool b_RRC_TaskReceiverOn:=TRUE;
    PERS bool b_RRC_TaskSenderOn:=TRUE;
    !
    PERS bool b_RRC_CtrlWaitForJob:=TRUE;
    PERS bool b_RRC_CtrlHamModOn:=FALSE;
    PERS bool b_RRC_CtrlInUse:=FALSE;
    PERS bool b_RRC_AutoIPAddress:=TRUE;
    PERS bool b_RRC_VirtualCustomPorts:=FALSE;
    !
    ! Channels
    PERS bool b_RRC_Com{n_RRC_NumOfCha}:=[TRUE,FALSE,FALSE,FALSE];
    PERS bool b_RRC_SIDCheck{n_RRC_NumOfCha}:=[TRUE,FALSE,FALSE,FALSE];
    PERS bool b_RRC_SIDErrorStop{n_RRC_NumOfCha}:=[FALSE,FALSE,FALSE,FALSE];
    PERS bool b_RRC_LogPro{n_RRC_NumOfCha}:=[FALSE,FALSE,FALSE,FALSE];
    !
    ! Client information
    PERS bool b_RRC_PPMain:=TRUE;
    !
    ! Activate or deactivate a event log message
    PERS bool b_RRC_EvLogReadAndUnpackTime:=FALSE;
    PERS bool b_RRC_EvLogPackAndSendTime:=FALSE;
    PERS bool b_RRC_EvLogMsgInUntilMsgOutTime:=FALSE;
    !
    ! Temporary to measure the feedback loop
    PERS bool b_RRC_FeedbackOut:=TRUE;

    !************************************************
    ! Declaration :     num
    !************************************************
    !
    !* PERS num n_RRC_WritePtrSenBufRob1:=1;
    PERS num n_RRC_WritePtrSenBufCtrl{n_RRC_NumOfCha}:=[0,0,0,0];
    PERS num n_RRC_WritePtrSenBufRob{n_RRC_NumOfCha}:=[7,0,0,0];
    !* PERS num n_RRC_SIDMax:=8388608;
    PERS num n_RRC_SIDMax:=1000000;
    !
    PERS num n_RRC_R1_ChaNr:=1;
    PERS num n_RRC_R2_ChaNr:=2;
    PERS num n_RRC_R3_ChaNr:=3;
    PERS num n_RRC_R4_ChaNr:=4;
    !
    PERS num n_RRC_SocketPortRec{n_RRC_NumOfCha}:=[30101,30102,30103,30104];
    PERS num n_RRC_SocketPortSen{n_RRC_NumOfCha}:=[30201,30202,30203,30204];
    !
    PERS num n_RRC_TimeTaskLiAll:=0.1;
    PERS num n_RRC_TimeTPMsg:=0.5;
    !
    PERS num n_RRC_ProtocolVersion:=2;

    !************************************************
    ! Declaration :     string
    !************************************************
    !
    PERS string n_RRC_Version:="v1.1.0";
    !
    PERS string st_RRC_CurCtrlJob:="RRC";
    PERS string st_RRC_JobForCtrl:="r_A031_HamMod";
    !
    PERS string st_RRC_IP_Address:="127.0.0.1";
    PERS string st_RRC_IP_AddressVC:="127.0.0.1";
    PERS string st_RRC_IP_AddressMan:="192.168.125.1";
    !
    ! System data
    PERS string st_RRC_SerialNr:="VIRTUAL_USE";
    PERS string st_RRC_SoftwareVersion:="ROBOTWARE_6.14.0139";
    PERS string st_RRC_RobotWare:="6.14.00.01";
    PERS string st_RRC_ControllerID:="VC";
    PERS string st_RRC_WAN_IP:="VC";
    PERS string st_RRC_ControllerLang:="en";
    PERS string st_RRC_SystemName:="vIRB4600-40-2.55-RW11";

    !************************************************
    ! Declaration :     tasklist
    !************************************************
    !
    PERS tasks tl_RRC_All{7}:=[["T_CTRL"],["T_RX"],["T_TX"],["T_ROB1"],[""],[""],[""]];

    !************************************************
    ! Declaration :     syncident
    !************************************************
    !
    VAR syncident id_RRC_MainSta;
    VAR syncident id_RRC_MainEnd;
    !
    VAR syncident id_RRC_InitSta;
    VAR syncident id_RRC_InitCtrl;
    VAR syncident id_RRC_InitEnd;

    !************************************************
    ! Declaration :     RRC_Channel
    !************************************************
    !
    PERS RRC_Channel ch_RRC_Channels:=[["T_ROB1",1],["T_ROB2",2],["T_ROB3",3],["T_ROB4",4]];

    !************************************************
    ! Declaration :     RRC_buffer_msg
    !************************************************
    !
    ! Receiver buffer for controller
    PERS RRC_buffer_msg bm_RRC_RecBufferCtrl{n_RRC_NumOfCha,10}:=[
    [[[0,0,0,"",0,0,"",0,0,0,"",0,"",0,"",0,"",0,"",0,"",0,"",0,"",0,0,0,0,0,0,0,0,0,0,0,0,0,0,0,0,0,0,0,0,0,0,0,0,0,0,0,0,0,0,0,0,0,0,0,0,0],FALSE],
    [[0,0,0,"",0,0,"",0,0,0,"",0,"",0,"",0,"",0,"",0,"",0,"",0,"",0,0,0,0,0,0,0,0,0,0,0,0,0,0,0,0,0,0,0,0,0,0,0,0,0,0,0,0,0,0,0,0,0,0,0,0,0],FALSE],
    [[0,0,0,"",0,0,"",0,0,0,"",0,"",0,"",0,"",0,"",0,"",0,"",0,"",0,0,0,0,0,0,0,0,0,0,0,0,0,0,0,0,0,0,0,0,0,0,0,0,0,0,0,0,0,0,0,0,0,0,0,0,0],FALSE],
    [[0,0,0,"",0,0,"",0,0,0,"",0,"",0,"",0,"",0,"",0,"",0,"",0,"",0,0,0,0,0,0,0,0,0,0,0,0,0,0,0,0,0,0,0,0,0,0,0,0,0,0,0,0,0,0,0,0,0,0,0,0,0],FALSE],
    [[0,0,0,"",0,0,"",0,0,0,"",0,"",0,"",0,"",0,"",0,"",0,"",0,"",0,0,0,0,0,0,0,0,0,0,0,0,0,0,0,0,0,0,0,0,0,0,0,0,0,0,0,0,0,0,0,0,0,0,0,0,0],FALSE],
    [[0,0,0,"",0,0,"",0,0,0,"",0,"",0,"",0,"",0,"",0,"",0,"",0,"",0,0,0,0,0,0,0,0,0,0,0,0,0,0,0,0,0,0,0,0,0,0,0,0,0,0,0,0,0,0,0,0,0,0,0,0,0],FALSE],
    [[0,0,0,"",0,0,"",0,0,0,"",0,"",0,"",0,"",0,"",0,"",0,"",0,"",0,0,0,0,0,0,0,0,0,0,0,0,0,0,0,0,0,0,0,0,0,0,0,0,0,0,0,0,0,0,0,0,0,0,0,0,0],FALSE],
    [[0,0,0,"",0,0,"",0,0,0,"",0,"",0,"",0,"",0,"",0,"",0,"",0,"",0,0,0,0,0,0,0,0,0,0,0,0,0,0,0,0,0,0,0,0,0,0,0,0,0,0,0,0,0,0,0,0,0,0,0,0,0],FALSE],
    [[0,0,0,"",0,0,"",0,0,0,"",0,"",0,"",0,"",0,"",0,"",0,"",0,"",0,0,0,0,0,0,0,0,0,0,0,0,0,0,0,0,0,0,0,0,0,0,0,0,0,0,0,0,0,0,0,0,0,0,0,0,0],FALSE],
    [[0,0,0,"",0,0,"",0,0,0,"",0,"",0,"",0,"",0,"",0,"",0,"",0,"",0,0,0,0,0,0,0,0,0,0,0,0,0,0,0,0,0,0,0,0,0,0,0,0,0,0,0,0,0,0,0,0,0,0,0,0,0],FALSE]],

    [[[0,0,0,"",0,0,"",0,0,0,"",0,"",0,"",0,"",0,"",0,"",0,"",0,"",0,0,0,0,0,0,0,0,0,0,0,0,0,0,0,0,0,0,0,0,0,0,0,0,0,0,0,0,0,0,0,0,0,0,0,0,0],FALSE],
    [[0,0,0,"",0,0,"",0,0,0,"",0,"",0,"",0,"",0,"",0,"",0,"",0,"",0,0,0,0,0,0,0,0,0,0,0,0,0,0,0,0,0,0,0,0,0,0,0,0,0,0,0,0,0,0,0,0,0,0,0,0,0],FALSE],
    [[0,0,0,"",0,0,"",0,0,0,"",0,"",0,"",0,"",0,"",0,"",0,"",0,"",0,0,0,0,0,0,0,0,0,0,0,0,0,0,0,0,0,0,0,0,0,0,0,0,0,0,0,0,0,0,0,0,0,0,0,0,0],FALSE],
    [[0,0,0,"",0,0,"",0,0,0,"",0,"",0,"",0,"",0,"",0,"",0,"",0,"",0,0,0,0,0,0,0,0,0,0,0,0,0,0,0,0,0,0,0,0,0,0,0,0,0,0,0,0,0,0,0,0,0,0,0,0,0],FALSE],
    [[0,0,0,"",0,0,"",0,0,0,"",0,"",0,"",0,"",0,"",0,"",0,"",0,"",0,0,0,0,0,0,0,0,0,0,0,0,0,0,0,0,0,0,0,0,0,0,0,0,0,0,0,0,0,0,0,0,0,0,0,0,0],FALSE],
    [[0,0,0,"",0,0,"",0,0,0,"",0,"",0,"",0,"",0,"",0,"",0,"",0,"",0,0,0,0,0,0,0,0,0,0,0,0,0,0,0,0,0,0,0,0,0,0,0,0,0,0,0,0,0,0,0,0,0,0,0,0,0],FALSE],
    [[0,0,0,"",0,0,"",0,0,0,"",0,"",0,"",0,"",0,"",0,"",0,"",0,"",0,0,0,0,0,0,0,0,0,0,0,0,0,0,0,0,0,0,0,0,0,0,0,0,0,0,0,0,0,0,0,0,0,0,0,0,0],FALSE],
    [[0,0,0,"",0,0,"",0,0,0,"",0,"",0,"",0,"",0,"",0,"",0,"",0,"",0,0,0,0,0,0,0,0,0,0,0,0,0,0,0,0,0,0,0,0,0,0,0,0,0,0,0,0,0,0,0,0,0,0,0,0,0],FALSE],
    [[0,0,0,"",0,0,"",0,0,0,"",0,"",0,"",0,"",0,"",0,"",0,"",0,"",0,0,0,0,0,0,0,0,0,0,0,0,0,0,0,0,0,0,0,0,0,0,0,0,0,0,0,0,0,0,0,0,0,0,0,0,0],FALSE],
    [[0,0,0,"",0,0,"",0,0,0,"",0,"",0,"",0,"",0,"",0,"",0,"",0,"",0,0,0,0,0,0,0,0,0,0,0,0,0,0,0,0,0,0,0,0,0,0,0,0,0,0,0,0,0,0,0,0,0,0,0,0,0],FALSE]],

    [[[0,0,0,"",0,0,"",0,0,0,"",0,"",0,"",0,"",0,"",0,"",0,"",0,"",0,0,0,0,0,0,0,0,0,0,0,0,0,0,0,0,0,0,0,0,0,0,0,0,0,0,0,0,0,0,0,0,0,0,0,0,0],FALSE],
    [[0,0,0,"",0,0,"",0,0,0,"",0,"",0,"",0,"",0,"",0,"",0,"",0,"",0,0,0,0,0,0,0,0,0,0,0,0,0,0,0,0,0,0,0,0,0,0,0,0,0,0,0,0,0,0,0,0,0,0,0,0,0],FALSE],
    [[0,0,0,"",0,0,"",0,0,0,"",0,"",0,"",0,"",0,"",0,"",0,"",0,"",0,0,0,0,0,0,0,0,0,0,0,0,0,0,0,0,0,0,0,0,0,0,0,0,0,0,0,0,0,0,0,0,0,0,0,0,0],FALSE],
    [[0,0,0,"",0,0,"",0,0,0,"",0,"",0,"",0,"",0,"",0,"",0,"",0,"",0,0,0,0,0,0,0,0,0,0,0,0,0,0,0,0,0,0,0,0,0,0,0,0,0,0,0,0,0,0,0,0,0,0,0,0,0],FALSE],
    [[0,0,0,"",0,0,"",0,0,0,"",0,"",0,"",0,"",0,"",0,"",0,"",0,"",0,0,0,0,0,0,0,0,0,0,0,0,0,0,0,0,0,0,0,0,0,0,0,0,0,0,0,0,0,0,0,0,0,0,0,0,0],FALSE],
    [[0,0,0,"",0,0,"",0,0,0,"",0,"",0,"",0,"",0,"",0,"",0,"",0,"",0,0,0,0,0,0,0,0,0,0,0,0,0,0,0,0,0,0,0,0,0,0,0,0,0,0,0,0,0,0,0,0,0,0,0,0,0],FALSE],
    [[0,0,0,"",0,0,"",0,0,0,"",0,"",0,"",0,"",0,"",0,"",0,"",0,"",0,0,0,0,0,0,0,0,0,0,0,0,0,0,0,0,0,0,0,0,0,0,0,0,0,0,0,0,0,0,0,0,0,0,0,0,0],FALSE],
    [[0,0,0,"",0,0,"",0,0,0,"",0,"",0,"",0,"",0,"",0,"",0,"",0,"",0,0,0,0,0,0,0,0,0,0,0,0,0,0,0,0,0,0,0,0,0,0,0,0,0,0,0,0,0,0,0,0,0,0,0,0,0],FALSE],
    [[0,0,0,"",0,0,"",0,0,0,"",0,"",0,"",0,"",0,"",0,"",0,"",0,"",0,0,0,0,0,0,0,0,0,0,0,0,0,0,0,0,0,0,0,0,0,0,0,0,0,0,0,0,0,0,0,0,0,0,0,0,0],FALSE],
    [[0,0,0,"",0,0,"",0,0,0,"",0,"",0,"",0,"",0,"",0,"",0,"",0,"",0,0,0,0,0,0,0,0,0,0,0,0,0,0,0,0,0,0,0,0,0,0,0,0,0,0,0,0,0,0,0,0,0,0,0,0,0],FALSE]],

    [[[0,0,0,"",0,0,"",0,0,0,"",0,"",0,"",0,"",0,"",0,"",0,"",0,"",0,0,0,0,0,0,0,0,0,0,0,0,0,0,0,0,0,0,0,0,0,0,0,0,0,0,0,0,0,0,0,0,0,0,0,0,0],FALSE],
    [[0,0,0,"",0,0,"",0,0,0,"",0,"",0,"",0,"",0,"",0,"",0,"",0,"",0,0,0,0,0,0,0,0,0,0,0,0,0,0,0,0,0,0,0,0,0,0,0,0,0,0,0,0,0,0,0,0,0,0,0,0,0],FALSE],
    [[0,0,0,"",0,0,"",0,0,0,"",0,"",0,"",0,"",0,"",0,"",0,"",0,"",0,0,0,0,0,0,0,0,0,0,0,0,0,0,0,0,0,0,0,0,0,0,0,0,0,0,0,0,0,0,0,0,0,0,0,0,0],FALSE],
    [[0,0,0,"",0,0,"",0,0,0,"",0,"",0,"",0,"",0,"",0,"",0,"",0,"",0,0,0,0,0,0,0,0,0,0,0,0,0,0,0,0,0,0,0,0,0,0,0,0,0,0,0,0,0,0,0,0,0,0,0,0,0],FALSE],
    [[0,0,0,"",0,0,"",0,0,0,"",0,"",0,"",0,"",0,"",0,"",0,"",0,"",0,0,0,0,0,0,0,0,0,0,0,0,0,0,0,0,0,0,0,0,0,0,0,0,0,0,0,0,0,0,0,0,0,0,0,0,0],FALSE],
    [[0,0,0,"",0,0,"",0,0,0,"",0,"",0,"",0,"",0,"",0,"",0,"",0,"",0,0,0,0,0,0,0,0,0,0,0,0,0,0,0,0,0,0,0,0,0,0,0,0,0,0,0,0,0,0,0,0,0,0,0,0,0],FALSE],
    [[0,0,0,"",0,0,"",0,0,0,"",0,"",0,"",0,"",0,"",0,"",0,"",0,"",0,0,0,0,0,0,0,0,0,0,0,0,0,0,0,0,0,0,0,0,0,0,0,0,0,0,0,0,0,0,0,0,0,0,0,0,0],FALSE],
    [[0,0,0,"",0,0,"",0,0,0,"",0,"",0,"",0,"",0,"",0,"",0,"",0,"",0,0,0,0,0,0,0,0,0,0,0,0,0,0,0,0,0,0,0,0,0,0,0,0,0,0,0,0,0,0,0,0,0,0,0,0,0],FALSE],
    [[0,0,0,"",0,0,"",0,0,0,"",0,"",0,"",0,"",0,"",0,"",0,"",0,"",0,0,0,0,0,0,0,0,0,0,0,0,0,0,0,0,0,0,0,0,0,0,0,0,0,0,0,0,0,0,0,0,0,0,0,0,0],FALSE],
    [[0,0,0,"",0,0,"",0,0,0,"",0,"",0,"",0,"",0,"",0,"",0,"",0,"",0,0,0,0,0,0,0,0,0,0,0,0,0,0,0,0,0,0,0,0,0,0,0,0,0,0,0,0,0,0,0,0,0,0,0,0,0],FALSE]]];

    !
    ! Receiver buffer for robots
    PERS RRC_buffer_msg bm_RRC_RecBufferRob{n_RRC_NumOfCha,10}:=[
    [[[1,0,15,"r_RRC_GetJoints",1,0,"",0,0,0,"",0,"",0,"",0,"",0,"",0,"",0,"",0,"",0,0,0,0,0,0,0,0,0,0,0,0,0,0,0,0,0,0,0,0,0,0,0,0,0,0,0,0,0,0,0,0,0,0,0,0,0],FALSE],
    [[1,0,15,"r_RRC_GetJoints",1,0,"",0,0,0,"",0,"",0,"",0,"",0,"",0,"",0,"",0,"",0,0,0,0,0,0,0,0,0,0,0,0,0,0,0,0,0,0,0,0,0,0,0,0,0,0,0,0,0,0,0,0,0,0,0,0,0],FALSE],
    [[1,0,15,"r_RRC_GetJoints",1,0,"",0,0,0,"",0,"",0,"",0,"",0,"",0,"",0,"",0,"",0,0,0,0,0,0,0,0,0,0,0,0,0,0,0,0,0,0,0,0,0,0,0,0,0,0,0,0,0,0,0,0,0,0,0,0,0],FALSE],
    [[1,0,15,"r_RRC_GetJoints",1,0,"",0,0,0,"",0,"",0,"",0,"",0,"",0,"",0,"",0,"",0,0,0,0,0,0,0,0,0,0,0,0,0,0,0,0,0,0,0,0,0,0,0,0,0,0,0,0,0,0,0,0,0,0,0,0,0],FALSE],
    [[1,0,15,"r_RRC_GetJoints",1,0,"",0,0,0,"",0,"",0,"",0,"",0,"",0,"",0,"",0,"",0,0,0,0,0,0,0,0,0,0,0,0,0,0,0,0,0,0,0,0,0,0,0,0,0,0,0,0,0,0,0,0,0,0,0,0,0],FALSE],
    [[1,0,15,"r_RRC_GetJoints",1,0,"",0,0,0,"",0,"",0,"",0,"",0,"",0,"",0,"",0,"",0,0,0,0,0,0,0,0,0,0,0,0,0,0,0,0,0,0,0,0,0,0,0,0,0,0,0,0,0,0,0,0,0,0,0,0,0],FALSE],
    [[1,0,15,"r_RRC_GetJoints",1,0,"",0,0,0,"",0,"",0,"",0,"",0,"",0,"",0,"",0,"",0,0,0,0,0,0,0,0,0,0,0,0,0,0,0,0,0,0,0,0,0,0,0,0,0,0,0,0,0,0,0,0,0,0,0,0,0],FALSE],
    [[1,0,15,"r_RRC_GetJoints",1,0,"",0,0,0,"",0,"",0,"",0,"",0,"",0,"",0,"",0,"",0,0,0,0,0,0,0,0,0,0,0,0,0,0,0,0,0,0,0,0,0,0,0,0,0,0,0,0,0,0,0,0,0,0,0,0,0],FALSE],
    [[1,0,15,"r_RRC_GetJoints",1,0,"",0,0,0,"",0,"",0,"",0,"",0,"",0,"",0,"",0,"",0,0,0,0,0,0,0,0,0,0,0,0,0,0,0,0,0,0,0,0,0,0,0,0,0,0,0,0,0,0,0,0,0,0,0,0,0],FALSE],
    [[1,0,15,"r_RRC_GetJoints",1,0,"",0,0,0,"",0,"",0,"",0,"",0,"",0,"",0,"",0,"",0,0,0,0,0,0,0,0,0,0,0,0,0,0,0,0,0,0,0,0,0,0,0,0,0,0,0,0,0,0,0,0,0,0,0,0,0],FALSE]],

    [[[0,0,0,"",0,0,"",0,0,0,"",0,"",0,"",0,"",0,"",0,"",0,"",0,"",0,0,0,0,0,0,0,0,0,0,0,0,0,0,0,0,0,0,0,0,0,0,0,0,0,0,0,0,0,0,0,0,0,0,0,0,0],FALSE],
    [[0,0,0,"",0,0,"",0,0,0,"",0,"",0,"",0,"",0,"",0,"",0,"",0,"",0,0,0,0,0,0,0,0,0,0,0,0,0,0,0,0,0,0,0,0,0,0,0,0,0,0,0,0,0,0,0,0,0,0,0,0,0],FALSE],
    [[0,0,0,"",0,0,"",0,0,0,"",0,"",0,"",0,"",0,"",0,"",0,"",0,"",0,0,0,0,0,0,0,0,0,0,0,0,0,0,0,0,0,0,0,0,0,0,0,0,0,0,0,0,0,0,0,0,0,0,0,0,0],FALSE],
    [[0,0,0,"",0,0,"",0,0,0,"",0,"",0,"",0,"",0,"",0,"",0,"",0,"",0,0,0,0,0,0,0,0,0,0,0,0,0,0,0,0,0,0,0,0,0,0,0,0,0,0,0,0,0,0,0,0,0,0,0,0,0],FALSE],
    [[0,0,0,"",0,0,"",0,0,0,"",0,"",0,"",0,"",0,"",0,"",0,"",0,"",0,0,0,0,0,0,0,0,0,0,0,0,0,0,0,0,0,0,0,0,0,0,0,0,0,0,0,0,0,0,0,0,0,0,0,0,0],FALSE],
    [[0,0,0,"",0,0,"",0,0,0,"",0,"",0,"",0,"",0,"",0,"",0,"",0,"",0,0,0,0,0,0,0,0,0,0,0,0,0,0,0,0,0,0,0,0,0,0,0,0,0,0,0,0,0,0,0,0,0,0,0,0,0],FALSE],
    [[0,0,0,"",0,0,"",0,0,0,"",0,"",0,"",0,"",0,"",0,"",0,"",0,"",0,0,0,0,0,0,0,0,0,0,0,0,0,0,0,0,0,0,0,0,0,0,0,0,0,0,0,0,0,0,0,0,0,0,0,0,0],FALSE],
    [[0,0,0,"",0,0,"",0,0,0,"",0,"",0,"",0,"",0,"",0,"",0,"",0,"",0,0,0,0,0,0,0,0,0,0,0,0,0,0,0,0,0,0,0,0,0,0,0,0,0,0,0,0,0,0,0,0,0,0,0,0,0],FALSE],
    [[0,0,0,"",0,0,"",0,0,0,"",0,"",0,"",0,"",0,"",0,"",0,"",0,"",0,0,0,0,0,0,0,0,0,0,0,0,0,0,0,0,0,0,0,0,0,0,0,0,0,0,0,0,0,0,0,0,0,0,0,0,0],FALSE],
    [[0,0,0,"",0,0,"",0,0,0,"",0,"",0,"",0,"",0,"",0,"",0,"",0,"",0,0,0,0,0,0,0,0,0,0,0,0,0,0,0,0,0,0,0,0,0,0,0,0,0,0,0,0,0,0,0,0,0,0,0,0,0],FALSE]],

    [[[0,0,0,"",0,0,"",0,0,0,"",0,"",0,"",0,"",0,"",0,"",0,"",0,"",0,0,0,0,0,0,0,0,0,0,0,0,0,0,0,0,0,0,0,0,0,0,0,0,0,0,0,0,0,0,0,0,0,0,0,0,0],FALSE],
    [[0,0,0,"",0,0,"",0,0,0,"",0,"",0,"",0,"",0,"",0,"",0,"",0,"",0,0,0,0,0,0,0,0,0,0,0,0,0,0,0,0,0,0,0,0,0,0,0,0,0,0,0,0,0,0,0,0,0,0,0,0,0],FALSE],
    [[0,0,0,"",0,0,"",0,0,0,"",0,"",0,"",0,"",0,"",0,"",0,"",0,"",0,0,0,0,0,0,0,0,0,0,0,0,0,0,0,0,0,0,0,0,0,0,0,0,0,0,0,0,0,0,0,0,0,0,0,0,0],FALSE],
    [[0,0,0,"",0,0,"",0,0,0,"",0,"",0,"",0,"",0,"",0,"",0,"",0,"",0,0,0,0,0,0,0,0,0,0,0,0,0,0,0,0,0,0,0,0,0,0,0,0,0,0,0,0,0,0,0,0,0,0,0,0,0],FALSE],
    [[0,0,0,"",0,0,"",0,0,0,"",0,"",0,"",0,"",0,"",0,"",0,"",0,"",0,0,0,0,0,0,0,0,0,0,0,0,0,0,0,0,0,0,0,0,0,0,0,0,0,0,0,0,0,0,0,0,0,0,0,0,0],FALSE],
    [[0,0,0,"",0,0,"",0,0,0,"",0,"",0,"",0,"",0,"",0,"",0,"",0,"",0,0,0,0,0,0,0,0,0,0,0,0,0,0,0,0,0,0,0,0,0,0,0,0,0,0,0,0,0,0,0,0,0,0,0,0,0],FALSE],
    [[0,0,0,"",0,0,"",0,0,0,"",0,"",0,"",0,"",0,"",0,"",0,"",0,"",0,0,0,0,0,0,0,0,0,0,0,0,0,0,0,0,0,0,0,0,0,0,0,0,0,0,0,0,0,0,0,0,0,0,0,0,0],FALSE],
    [[0,0,0,"",0,0,"",0,0,0,"",0,"",0,"",0,"",0,"",0,"",0,"",0,"",0,0,0,0,0,0,0,0,0,0,0,0,0,0,0,0,0,0,0,0,0,0,0,0,0,0,0,0,0,0,0,0,0,0,0,0,0],FALSE],
    [[0,0,0,"",0,0,"",0,0,0,"",0,"",0,"",0,"",0,"",0,"",0,"",0,"",0,0,0,0,0,0,0,0,0,0,0,0,0,0,0,0,0,0,0,0,0,0,0,0,0,0,0,0,0,0,0,0,0,0,0,0,0],FALSE],
    [[0,0,0,"",0,0,"",0,0,0,"",0,"",0,"",0,"",0,"",0,"",0,"",0,"",0,0,0,0,0,0,0,0,0,0,0,0,0,0,0,0,0,0,0,0,0,0,0,0,0,0,0,0,0,0,0,0,0,0,0,0,0],FALSE]],

    [[[0,0,0,"",0,0,"",0,0,0,"",0,"",0,"",0,"",0,"",0,"",0,"",0,"",0,0,0,0,0,0,0,0,0,0,0,0,0,0,0,0,0,0,0,0,0,0,0,0,0,0,0,0,0,0,0,0,0,0,0,0,0],FALSE],
    [[0,0,0,"",0,0,"",0,0,0,"",0,"",0,"",0,"",0,"",0,"",0,"",0,"",0,0,0,0,0,0,0,0,0,0,0,0,0,0,0,0,0,0,0,0,0,0,0,0,0,0,0,0,0,0,0,0,0,0,0,0,0],FALSE],
    [[0,0,0,"",0,0,"",0,0,0,"",0,"",0,"",0,"",0,"",0,"",0,"",0,"",0,0,0,0,0,0,0,0,0,0,0,0,0,0,0,0,0,0,0,0,0,0,0,0,0,0,0,0,0,0,0,0,0,0,0,0,0],FALSE],
    [[0,0,0,"",0,0,"",0,0,0,"",0,"",0,"",0,"",0,"",0,"",0,"",0,"",0,0,0,0,0,0,0,0,0,0,0,0,0,0,0,0,0,0,0,0,0,0,0,0,0,0,0,0,0,0,0,0,0,0,0,0,0],FALSE],
    [[0,0,0,"",0,0,"",0,0,0,"",0,"",0,"",0,"",0,"",0,"",0,"",0,"",0,0,0,0,0,0,0,0,0,0,0,0,0,0,0,0,0,0,0,0,0,0,0,0,0,0,0,0,0,0,0,0,0,0,0,0,0],FALSE],
    [[0,0,0,"",0,0,"",0,0,0,"",0,"",0,"",0,"",0,"",0,"",0,"",0,"",0,0,0,0,0,0,0,0,0,0,0,0,0,0,0,0,0,0,0,0,0,0,0,0,0,0,0,0,0,0,0,0,0,0,0,0,0],FALSE],
    [[0,0,0,"",0,0,"",0,0,0,"",0,"",0,"",0,"",0,"",0,"",0,"",0,"",0,0,0,0,0,0,0,0,0,0,0,0,0,0,0,0,0,0,0,0,0,0,0,0,0,0,0,0,0,0,0,0,0,0,0,0,0],FALSE],
    [[0,0,0,"",0,0,"",0,0,0,"",0,"",0,"",0,"",0,"",0,"",0,"",0,"",0,0,0,0,0,0,0,0,0,0,0,0,0,0,0,0,0,0,0,0,0,0,0,0,0,0,0,0,0,0,0,0,0,0,0,0,0],FALSE],
    [[0,0,0,"",0,0,"",0,0,0,"",0,"",0,"",0,"",0,"",0,"",0,"",0,"",0,0,0,0,0,0,0,0,0,0,0,0,0,0,0,0,0,0,0,0,0,0,0,0,0,0,0,0,0,0,0,0,0,0,0,0,0],FALSE],
    [[0,0,0,"",0,0,"",0,0,0,"",0,"",0,"",0,"",0,"",0,"",0,"",0,"",0,0,0,0,0,0,0,0,0,0,0,0,0,0,0,0,0,0,0,0,0,0,0,0,0,0,0,0,0,0,0,0,0,0,0,0,0],FALSE]]];

    !
    ! Sender buffer for controller
    PERS RRC_buffer_msg bm_RRC_SenBufferCtrl{n_RRC_NumOfCha,10}:=[
    [[[0,0,0,"",0,0,"",0,0,0,"",0,"",0,"",0,"",0,"",0,"",0,"",0,"",0,0,0,0,0,0,0,0,0,0,0,0,0,0,0,0,0,0,0,0,0,0,0,0,0,0,0,0,0,0,0,0,0,0,0,0,0],FALSE],
    [[0,0,0,"",0,0,"",0,0,0,"",0,"",0,"",0,"",0,"",0,"",0,"",0,"",0,0,0,0,0,0,0,0,0,0,0,0,0,0,0,0,0,0,0,0,0,0,0,0,0,0,0,0,0,0,0,0,0,0,0,0,0],FALSE],
    [[0,0,0,"",0,0,"",0,0,0,"",0,"",0,"",0,"",0,"",0,"",0,"",0,"",0,0,0,0,0,0,0,0,0,0,0,0,0,0,0,0,0,0,0,0,0,0,0,0,0,0,0,0,0,0,0,0,0,0,0,0,0],FALSE],
    [[0,0,0,"",0,0,"",0,0,0,"",0,"",0,"",0,"",0,"",0,"",0,"",0,"",0,0,0,0,0,0,0,0,0,0,0,0,0,0,0,0,0,0,0,0,0,0,0,0,0,0,0,0,0,0,0,0,0,0,0,0,0],FALSE],
    [[0,0,0,"",0,0,"",0,0,0,"",0,"",0,"",0,"",0,"",0,"",0,"",0,"",0,0,0,0,0,0,0,0,0,0,0,0,0,0,0,0,0,0,0,0,0,0,0,0,0,0,0,0,0,0,0,0,0,0,0,0,0],FALSE],
    [[0,0,0,"",0,0,"",0,0,0,"",0,"",0,"",0,"",0,"",0,"",0,"",0,"",0,0,0,0,0,0,0,0,0,0,0,0,0,0,0,0,0,0,0,0,0,0,0,0,0,0,0,0,0,0,0,0,0,0,0,0,0],FALSE],
    [[0,0,0,"",0,0,"",0,0,0,"",0,"",0,"",0,"",0,"",0,"",0,"",0,"",0,0,0,0,0,0,0,0,0,0,0,0,0,0,0,0,0,0,0,0,0,0,0,0,0,0,0,0,0,0,0,0,0,0,0,0,0],FALSE],
    [[0,0,0,"",0,0,"",0,0,0,"",0,"",0,"",0,"",0,"",0,"",0,"",0,"",0,0,0,0,0,0,0,0,0,0,0,0,0,0,0,0,0,0,0,0,0,0,0,0,0,0,0,0,0,0,0,0,0,0,0,0,0],FALSE],
    [[0,0,0,"",0,0,"",0,0,0,"",0,"",0,"",0,"",0,"",0,"",0,"",0,"",0,0,0,0,0,0,0,0,0,0,0,0,0,0,0,0,0,0,0,0,0,0,0,0,0,0,0,0,0,0,0,0,0,0,0,0,0],FALSE],
    [[0,0,0,"",0,0,"",0,0,0,"",0,"",0,"",0,"",0,"",0,"",0,"",0,"",0,0,0,0,0,0,0,0,0,0,0,0,0,0,0,0,0,0,0,0,0,0,0,0,0,0,0,0,0,0,0,0,0,0,0,0,0],FALSE]],

    [[[0,0,0,"",0,0,"",0,0,0,"",0,"",0,"",0,"",0,"",0,"",0,"",0,"",0,0,0,0,0,0,0,0,0,0,0,0,0,0,0,0,0,0,0,0,0,0,0,0,0,0,0,0,0,0,0,0,0,0,0,0,0],FALSE],
    [[0,0,0,"",0,0,"",0,0,0,"",0,"",0,"",0,"",0,"",0,"",0,"",0,"",0,0,0,0,0,0,0,0,0,0,0,0,0,0,0,0,0,0,0,0,0,0,0,0,0,0,0,0,0,0,0,0,0,0,0,0,0],FALSE],
    [[0,0,0,"",0,0,"",0,0,0,"",0,"",0,"",0,"",0,"",0,"",0,"",0,"",0,0,0,0,0,0,0,0,0,0,0,0,0,0,0,0,0,0,0,0,0,0,0,0,0,0,0,0,0,0,0,0,0,0,0,0,0],FALSE],
    [[0,0,0,"",0,0,"",0,0,0,"",0,"",0,"",0,"",0,"",0,"",0,"",0,"",0,0,0,0,0,0,0,0,0,0,0,0,0,0,0,0,0,0,0,0,0,0,0,0,0,0,0,0,0,0,0,0,0,0,0,0,0],FALSE],
    [[0,0,0,"",0,0,"",0,0,0,"",0,"",0,"",0,"",0,"",0,"",0,"",0,"",0,0,0,0,0,0,0,0,0,0,0,0,0,0,0,0,0,0,0,0,0,0,0,0,0,0,0,0,0,0,0,0,0,0,0,0,0],FALSE],
    [[0,0,0,"",0,0,"",0,0,0,"",0,"",0,"",0,"",0,"",0,"",0,"",0,"",0,0,0,0,0,0,0,0,0,0,0,0,0,0,0,0,0,0,0,0,0,0,0,0,0,0,0,0,0,0,0,0,0,0,0,0,0],FALSE],
    [[0,0,0,"",0,0,"",0,0,0,"",0,"",0,"",0,"",0,"",0,"",0,"",0,"",0,0,0,0,0,0,0,0,0,0,0,0,0,0,0,0,0,0,0,0,0,0,0,0,0,0,0,0,0,0,0,0,0,0,0,0,0],FALSE],
    [[0,0,0,"",0,0,"",0,0,0,"",0,"",0,"",0,"",0,"",0,"",0,"",0,"",0,0,0,0,0,0,0,0,0,0,0,0,0,0,0,0,0,0,0,0,0,0,0,0,0,0,0,0,0,0,0,0,0,0,0,0,0],FALSE],
    [[0,0,0,"",0,0,"",0,0,0,"",0,"",0,"",0,"",0,"",0,"",0,"",0,"",0,0,0,0,0,0,0,0,0,0,0,0,0,0,0,0,0,0,0,0,0,0,0,0,0,0,0,0,0,0,0,0,0,0,0,0,0],FALSE],
    [[0,0,0,"",0,0,"",0,0,0,"",0,"",0,"",0,"",0,"",0,"",0,"",0,"",0,0,0,0,0,0,0,0,0,0,0,0,0,0,0,0,0,0,0,0,0,0,0,0,0,0,0,0,0,0,0,0,0,0,0,0,0],FALSE]],

    [[[0,0,0,"",0,0,"",0,0,0,"",0,"",0,"",0,"",0,"",0,"",0,"",0,"",0,0,0,0,0,0,0,0,0,0,0,0,0,0,0,0,0,0,0,0,0,0,0,0,0,0,0,0,0,0,0,0,0,0,0,0,0],FALSE],
    [[0,0,0,"",0,0,"",0,0,0,"",0,"",0,"",0,"",0,"",0,"",0,"",0,"",0,0,0,0,0,0,0,0,0,0,0,0,0,0,0,0,0,0,0,0,0,0,0,0,0,0,0,0,0,0,0,0,0,0,0,0,0],FALSE],
    [[0,0,0,"",0,0,"",0,0,0,"",0,"",0,"",0,"",0,"",0,"",0,"",0,"",0,0,0,0,0,0,0,0,0,0,0,0,0,0,0,0,0,0,0,0,0,0,0,0,0,0,0,0,0,0,0,0,0,0,0,0,0],FALSE],
    [[0,0,0,"",0,0,"",0,0,0,"",0,"",0,"",0,"",0,"",0,"",0,"",0,"",0,0,0,0,0,0,0,0,0,0,0,0,0,0,0,0,0,0,0,0,0,0,0,0,0,0,0,0,0,0,0,0,0,0,0,0,0],FALSE],
    [[0,0,0,"",0,0,"",0,0,0,"",0,"",0,"",0,"",0,"",0,"",0,"",0,"",0,0,0,0,0,0,0,0,0,0,0,0,0,0,0,0,0,0,0,0,0,0,0,0,0,0,0,0,0,0,0,0,0,0,0,0,0],FALSE],
    [[0,0,0,"",0,0,"",0,0,0,"",0,"",0,"",0,"",0,"",0,"",0,"",0,"",0,0,0,0,0,0,0,0,0,0,0,0,0,0,0,0,0,0,0,0,0,0,0,0,0,0,0,0,0,0,0,0,0,0,0,0,0],FALSE],
    [[0,0,0,"",0,0,"",0,0,0,"",0,"",0,"",0,"",0,"",0,"",0,"",0,"",0,0,0,0,0,0,0,0,0,0,0,0,0,0,0,0,0,0,0,0,0,0,0,0,0,0,0,0,0,0,0,0,0,0,0,0,0],FALSE],
    [[0,0,0,"",0,0,"",0,0,0,"",0,"",0,"",0,"",0,"",0,"",0,"",0,"",0,0,0,0,0,0,0,0,0,0,0,0,0,0,0,0,0,0,0,0,0,0,0,0,0,0,0,0,0,0,0,0,0,0,0,0,0],FALSE],
    [[0,0,0,"",0,0,"",0,0,0,"",0,"",0,"",0,"",0,"",0,"",0,"",0,"",0,0,0,0,0,0,0,0,0,0,0,0,0,0,0,0,0,0,0,0,0,0,0,0,0,0,0,0,0,0,0,0,0,0,0,0,0],FALSE],
    [[0,0,0,"",0,0,"",0,0,0,"",0,"",0,"",0,"",0,"",0,"",0,"",0,"",0,0,0,0,0,0,0,0,0,0,0,0,0,0,0,0,0,0,0,0,0,0,0,0,0,0,0,0,0,0,0,0,0,0,0,0,0],FALSE]],

    [[[0,0,0,"",0,0,"",0,0,0,"",0,"",0,"",0,"",0,"",0,"",0,"",0,"",0,0,0,0,0,0,0,0,0,0,0,0,0,0,0,0,0,0,0,0,0,0,0,0,0,0,0,0,0,0,0,0,0,0,0,0,0],FALSE],
    [[0,0,0,"",0,0,"",0,0,0,"",0,"",0,"",0,"",0,"",0,"",0,"",0,"",0,0,0,0,0,0,0,0,0,0,0,0,0,0,0,0,0,0,0,0,0,0,0,0,0,0,0,0,0,0,0,0,0,0,0,0,0],FALSE],
    [[0,0,0,"",0,0,"",0,0,0,"",0,"",0,"",0,"",0,"",0,"",0,"",0,"",0,0,0,0,0,0,0,0,0,0,0,0,0,0,0,0,0,0,0,0,0,0,0,0,0,0,0,0,0,0,0,0,0,0,0,0,0],FALSE],
    [[0,0,0,"",0,0,"",0,0,0,"",0,"",0,"",0,"",0,"",0,"",0,"",0,"",0,0,0,0,0,0,0,0,0,0,0,0,0,0,0,0,0,0,0,0,0,0,0,0,0,0,0,0,0,0,0,0,0,0,0,0,0],FALSE],
    [[0,0,0,"",0,0,"",0,0,0,"",0,"",0,"",0,"",0,"",0,"",0,"",0,"",0,0,0,0,0,0,0,0,0,0,0,0,0,0,0,0,0,0,0,0,0,0,0,0,0,0,0,0,0,0,0,0,0,0,0,0,0],FALSE],
    [[0,0,0,"",0,0,"",0,0,0,"",0,"",0,"",0,"",0,"",0,"",0,"",0,"",0,0,0,0,0,0,0,0,0,0,0,0,0,0,0,0,0,0,0,0,0,0,0,0,0,0,0,0,0,0,0,0,0,0,0,0,0],FALSE],
    [[0,0,0,"",0,0,"",0,0,0,"",0,"",0,"",0,"",0,"",0,"",0,"",0,"",0,0,0,0,0,0,0,0,0,0,0,0,0,0,0,0,0,0,0,0,0,0,0,0,0,0,0,0,0,0,0,0,0,0,0,0,0],FALSE],
    [[0,0,0,"",0,0,"",0,0,0,"",0,"",0,"",0,"",0,"",0,"",0,"",0,"",0,0,0,0,0,0,0,0,0,0,0,0,0,0,0,0,0,0,0,0,0,0,0,0,0,0,0,0,0,0,0,0,0,0,0,0,0],FALSE],
    [[0,0,0,"",0,0,"",0,0,0,"",0,"",0,"",0,"",0,"",0,"",0,"",0,"",0,0,0,0,0,0,0,0,0,0,0,0,0,0,0,0,0,0,0,0,0,0,0,0,0,0,0,0,0,0,0,0,0,0,0,0,0],FALSE],
    [[0,0,0,"",0,0,"",0,0,0,"",0,"",0,"",0,"",0,"",0,"",0,"",0,"",0,0,0,0,0,0,0,0,0,0,0,0,0,0,0,0,0,0,0,0,0,0,0,0,0,0,0,0,0,0,0,0,0,0,0,0,0],FALSE]]];

    !
    ! Sender buffer for robots
    PERS RRC_buffer_msg bm_RRC_SenBufferRob{n_RRC_NumOfCha,10}:=[
    [[[0,0,0,"r_RRC_GetJoints",0,0,"Done",1,0,0,"",0,"",0,"",0,"",0,"",0,"",0,"",0,"",12,-24.4963,-17.8131,33.2614,-59.6898,-28.7042,56.3166,9E+9,9E+9,9E+9,9E+9,9E+9,9E+9,0,0,0,0,0,0,0,0,0,0,0,0,0,0,0,0,0,0,0,0,0,0,0,0],FALSE],
    [[0,0,0,"r_RRC_GetJoints",0,0,"Done",1,0,0,"",0,"",0,"",0,"",0,"",0,"",0,"",0,"",12,-24.4963,-17.8131,33.2614,-59.6898,-28.7042,56.3166,9E+9,9E+9,9E+9,9E+9,9E+9,9E+9,0,0,0,0,0,0,0,0,0,0,0,0,0,0,0,0,0,0,0,0,0,0,0,0],FALSE],
    [[0,0,0,"r_RRC_GetJoints",0,0,"Done",1,0,0,"",0,"",0,"",0,"",0,"",0,"",0,"",0,"",12,-24.4963,-17.8131,33.2614,-59.6898,-28.7042,56.3166,9E+9,9E+9,9E+9,9E+9,9E+9,9E+9,0,0,0,0,0,0,0,0,0,0,0,0,0,0,0,0,0,0,0,0,0,0,0,0],FALSE],
    [[0,0,0,"r_RRC_GetJoints",0,0,"Done",1,0,0,"",0,"",0,"",0,"",0,"",0,"",0,"",0,"",12,-24.4963,-17.8131,33.2614,-59.6898,-28.7042,56.3166,9E+9,9E+9,9E+9,9E+9,9E+9,9E+9,0,0,0,0,0,0,0,0,0,0,0,0,0,0,0,0,0,0,0,0,0,0,0,0],FALSE],
    [[0,0,0,"r_RRC_GetJoints",0,0,"Done",1,0,0,"",0,"",0,"",0,"",0,"",0,"",0,"",0,"",12,-24.4963,-17.8131,33.2614,-59.6898,-28.7042,56.3166,9E+9,9E+9,9E+9,9E+9,9E+9,9E+9,0,0,0,0,0,0,0,0,0,0,0,0,0,0,0,0,0,0,0,0,0,0,0,0],FALSE],
    [[0,0,0,"r_RRC_GetJoints",0,0,"Done",1,0,0,"",0,"",0,"",0,"",0,"",0,"",0,"",0,"",12,-24.4963,-17.8131,33.2614,-59.6898,-28.7042,56.3166,9E+9,9E+9,9E+9,9E+9,9E+9,9E+9,0,0,0,0,0,0,0,0,0,0,0,0,0,0,0,0,0,0,0,0,0,0,0,0],FALSE],
    [[0,0,0,"r_RRC_GetJoints",0,0,"Done",1,0,0,"",0,"",0,"",0,"",0,"",0,"",0,"",0,"",12,-24.4963,-17.8131,33.2614,-59.6898,-28.7042,56.3166,9E+9,9E+9,9E+9,9E+9,9E+9,9E+9,0,0,0,0,0,0,0,0,0,0,0,0,0,0,0,0,0,0,0,0,0,0,0,0],FALSE],
    [[0,0,0,"r_RRC_GetJoints",0,0,"Done",1,0,0,"",0,"",0,"",0,"",0,"",0,"",0,"",0,"",12,-24.4963,-17.8131,33.2614,-59.6898,-28.7042,56.3166,9E+9,9E+9,9E+9,9E+9,9E+9,9E+9,0,0,0,0,0,0,0,0,0,0,0,0,0,0,0,0,0,0,0,0,0,0,0,0],FALSE],
    [[0,0,0,"r_RRC_GetJoints",0,0,"Done",1,0,0,"",0,"",0,"",0,"",0,"",0,"",0,"",0,"",12,-24.4963,-17.8131,33.2614,-59.6898,-28.7042,56.3166,9E+9,9E+9,9E+9,9E+9,9E+9,9E+9,0,0,0,0,0,0,0,0,0,0,0,0,0,0,0,0,0,0,0,0,0,0,0,0],FALSE],
    [[0,0,0,"r_RRC_GetJoints",0,0,"Done",1,0,0,"",0,"",0,"",0,"",0,"",0,"",0,"",0,"",12,-24.4963,-17.8131,33.2614,-59.6898,-28.7042,56.3166,9E+9,9E+9,9E+9,9E+9,9E+9,9E+9,0,0,0,0,0,0,0,0,0,0,0,0,0,0,0,0,0,0,0,0,0,0,0,0],FALSE]],

    [[[0,0,0,"",0,0,"",0,0,0,"",0,"",0,"",0,"",0,"",0,"",0,"",0,"",0,0,0,0,0,0,0,0,0,0,0,0,0,0,0,0,0,0,0,0,0,0,0,0,0,0,0,0,0,0,0,0,0,0,0,0,0],FALSE],
    [[0,0,0,"",0,0,"",0,0,0,"",0,"",0,"",0,"",0,"",0,"",0,"",0,"",0,0,0,0,0,0,0,0,0,0,0,0,0,0,0,0,0,0,0,0,0,0,0,0,0,0,0,0,0,0,0,0,0,0,0,0,0],FALSE],
    [[0,0,0,"",0,0,"",0,0,0,"",0,"",0,"",0,"",0,"",0,"",0,"",0,"",0,0,0,0,0,0,0,0,0,0,0,0,0,0,0,0,0,0,0,0,0,0,0,0,0,0,0,0,0,0,0,0,0,0,0,0,0],FALSE],
    [[0,0,0,"",0,0,"",0,0,0,"",0,"",0,"",0,"",0,"",0,"",0,"",0,"",0,0,0,0,0,0,0,0,0,0,0,0,0,0,0,0,0,0,0,0,0,0,0,0,0,0,0,0,0,0,0,0,0,0,0,0,0],FALSE],
    [[0,0,0,"",0,0,"",0,0,0,"",0,"",0,"",0,"",0,"",0,"",0,"",0,"",0,0,0,0,0,0,0,0,0,0,0,0,0,0,0,0,0,0,0,0,0,0,0,0,0,0,0,0,0,0,0,0,0,0,0,0,0],FALSE],
    [[0,0,0,"",0,0,"",0,0,0,"",0,"",0,"",0,"",0,"",0,"",0,"",0,"",0,0,0,0,0,0,0,0,0,0,0,0,0,0,0,0,0,0,0,0,0,0,0,0,0,0,0,0,0,0,0,0,0,0,0,0,0],FALSE],
    [[0,0,0,"",0,0,"",0,0,0,"",0,"",0,"",0,"",0,"",0,"",0,"",0,"",0,0,0,0,0,0,0,0,0,0,0,0,0,0,0,0,0,0,0,0,0,0,0,0,0,0,0,0,0,0,0,0,0,0,0,0,0],FALSE],
    [[0,0,0,"",0,0,"",0,0,0,"",0,"",0,"",0,"",0,"",0,"",0,"",0,"",0,0,0,0,0,0,0,0,0,0,0,0,0,0,0,0,0,0,0,0,0,0,0,0,0,0,0,0,0,0,0,0,0,0,0,0,0],FALSE],
    [[0,0,0,"",0,0,"",0,0,0,"",0,"",0,"",0,"",0,"",0,"",0,"",0,"",0,0,0,0,0,0,0,0,0,0,0,0,0,0,0,0,0,0,0,0,0,0,0,0,0,0,0,0,0,0,0,0,0,0,0,0,0],FALSE],
    [[0,0,0,"",0,0,"",0,0,0,"",0,"",0,"",0,"",0,"",0,"",0,"",0,"",0,0,0,0,0,0,0,0,0,0,0,0,0,0,0,0,0,0,0,0,0,0,0,0,0,0,0,0,0,0,0,0,0,0,0,0,0],FALSE]],

    [[[0,0,0,"",0,0,"",0,0,0,"",0,"",0,"",0,"",0,"",0,"",0,"",0,"",0,0,0,0,0,0,0,0,0,0,0,0,0,0,0,0,0,0,0,0,0,0,0,0,0,0,0,0,0,0,0,0,0,0,0,0,0],FALSE],
    [[0,0,0,"",0,0,"",0,0,0,"",0,"",0,"",0,"",0,"",0,"",0,"",0,"",0,0,0,0,0,0,0,0,0,0,0,0,0,0,0,0,0,0,0,0,0,0,0,0,0,0,0,0,0,0,0,0,0,0,0,0,0],FALSE],
    [[0,0,0,"",0,0,"",0,0,0,"",0,"",0,"",0,"",0,"",0,"",0,"",0,"",0,0,0,0,0,0,0,0,0,0,0,0,0,0,0,0,0,0,0,0,0,0,0,0,0,0,0,0,0,0,0,0,0,0,0,0,0],FALSE],
    [[0,0,0,"",0,0,"",0,0,0,"",0,"",0,"",0,"",0,"",0,"",0,"",0,"",0,0,0,0,0,0,0,0,0,0,0,0,0,0,0,0,0,0,0,0,0,0,0,0,0,0,0,0,0,0,0,0,0,0,0,0,0],FALSE],
    [[0,0,0,"",0,0,"",0,0,0,"",0,"",0,"",0,"",0,"",0,"",0,"",0,"",0,0,0,0,0,0,0,0,0,0,0,0,0,0,0,0,0,0,0,0,0,0,0,0,0,0,0,0,0,0,0,0,0,0,0,0,0],FALSE],
    [[0,0,0,"",0,0,"",0,0,0,"",0,"",0,"",0,"",0,"",0,"",0,"",0,"",0,0,0,0,0,0,0,0,0,0,0,0,0,0,0,0,0,0,0,0,0,0,0,0,0,0,0,0,0,0,0,0,0,0,0,0,0],FALSE],
    [[0,0,0,"",0,0,"",0,0,0,"",0,"",0,"",0,"",0,"",0,"",0,"",0,"",0,0,0,0,0,0,0,0,0,0,0,0,0,0,0,0,0,0,0,0,0,0,0,0,0,0,0,0,0,0,0,0,0,0,0,0,0],FALSE],
    [[0,0,0,"",0,0,"",0,0,0,"",0,"",0,"",0,"",0,"",0,"",0,"",0,"",0,0,0,0,0,0,0,0,0,0,0,0,0,0,0,0,0,0,0,0,0,0,0,0,0,0,0,0,0,0,0,0,0,0,0,0,0],FALSE],
    [[0,0,0,"",0,0,"",0,0,0,"",0,"",0,"",0,"",0,"",0,"",0,"",0,"",0,0,0,0,0,0,0,0,0,0,0,0,0,0,0,0,0,0,0,0,0,0,0,0,0,0,0,0,0,0,0,0,0,0,0,0,0],FALSE],
    [[0,0,0,"",0,0,"",0,0,0,"",0,"",0,"",0,"",0,"",0,"",0,"",0,"",0,0,0,0,0,0,0,0,0,0,0,0,0,0,0,0,0,0,0,0,0,0,0,0,0,0,0,0,0,0,0,0,0,0,0,0,0],FALSE]],

    [[[0,0,0,"",0,0,"",0,0,0,"",0,"",0,"",0,"",0,"",0,"",0,"",0,"",0,0,0,0,0,0,0,0,0,0,0,0,0,0,0,0,0,0,0,0,0,0,0,0,0,0,0,0,0,0,0,0,0,0,0,0,0],FALSE],
    [[0,0,0,"",0,0,"",0,0,0,"",0,"",0,"",0,"",0,"",0,"",0,"",0,"",0,0,0,0,0,0,0,0,0,0,0,0,0,0,0,0,0,0,0,0,0,0,0,0,0,0,0,0,0,0,0,0,0,0,0,0,0],FALSE],
    [[0,0,0,"",0,0,"",0,0,0,"",0,"",0,"",0,"",0,"",0,"",0,"",0,"",0,0,0,0,0,0,0,0,0,0,0,0,0,0,0,0,0,0,0,0,0,0,0,0,0,0,0,0,0,0,0,0,0,0,0,0,0],FALSE],
    [[0,0,0,"",0,0,"",0,0,0,"",0,"",0,"",0,"",0,"",0,"",0,"",0,"",0,0,0,0,0,0,0,0,0,0,0,0,0,0,0,0,0,0,0,0,0,0,0,0,0,0,0,0,0,0,0,0,0,0,0,0,0],FALSE],
    [[0,0,0,"",0,0,"",0,0,0,"",0,"",0,"",0,"",0,"",0,"",0,"",0,"",0,0,0,0,0,0,0,0,0,0,0,0,0,0,0,0,0,0,0,0,0,0,0,0,0,0,0,0,0,0,0,0,0,0,0,0,0],FALSE],
    [[0,0,0,"",0,0,"",0,0,0,"",0,"",0,"",0,"",0,"",0,"",0,"",0,"",0,0,0,0,0,0,0,0,0,0,0,0,0,0,0,0,0,0,0,0,0,0,0,0,0,0,0,0,0,0,0,0,0,0,0,0,0],FALSE],
    [[0,0,0,"",0,0,"",0,0,0,"",0,"",0,"",0,"",0,"",0,"",0,"",0,"",0,0,0,0,0,0,0,0,0,0,0,0,0,0,0,0,0,0,0,0,0,0,0,0,0,0,0,0,0,0,0,0,0,0,0,0,0],FALSE],
    [[0,0,0,"",0,0,"",0,0,0,"",0,"",0,"",0,"",0,"",0,"",0,"",0,"",0,0,0,0,0,0,0,0,0,0,0,0,0,0,0,0,0,0,0,0,0,0,0,0,0,0,0,0,0,0,0,0,0,0,0,0,0],FALSE],
    [[0,0,0,"",0,0,"",0,0,0,"",0,"",0,"",0,"",0,"",0,"",0,"",0,"",0,0,0,0,0,0,0,0,0,0,0,0,0,0,0,0,0,0,0,0,0,0,0,0,0,0,0,0,0,0,0,0,0,0,0,0,0],FALSE],
    [[0,0,0,"",0,0,"",0,0,0,"",0,"",0,"",0,"",0,"",0,"",0,"",0,"",0,0,0,0,0,0,0,0,0,0,0,0,0,0,0,0,0,0,0,0,0,0,0,0,0,0,0,0,0,0,0,0,0,0,0,0,0],FALSE]]];

ENDMODULE

--- Backups/vIRB4600-40-2.55-RW11/RAPID/TASK2/SYSMOD/RRC_DataTask_Ctrl.sys ---
MODULE RRC_DataTask_Ctrl(SYSMODULE)
    !***********************************************************************************
    !
    ! ETH Zurich / Robotic Fabrication Lab
    ! HIB C 13 / Stefano-Franscini-Platz 1
    ! CH-8093 Zurich
    !
    !***********************************************************************************
    !
    ! PROJECT     :  RRC - Rapid Robot Communication
    !
    ! FUNCTION    :  Includ all Task specific Data's
    !
    ! AUTHOR      :  Philippe Fleischmann
    !
    ! EMAIL       :  rrc@arch.ethz.ch
    !
    ! HISTORY     :  2019.02.22
    !
    ! Copyright   :  ETH Zurich (CH) 2019
    !                - Philippe Fleischmann
    !                - Michael Lyrenmann
    !                - Gonzalo Casas
    !
    ! License     :  This code base is governed by an EULA (End-User License Agreement)
    !                which you have received together with the software.
    !                You are not allowed to use the software on a real robots
    !                without a signed EULA.
    !
    !                A copy of the EULA content is in the controller task (T_CTRL).
    !
    !***********************************************************************************

    !************************************************
    ! Declaration :     bool
    !************************************************
    !
    CONST bool b_RRC_Run:=TRUE;
    !
    TASK PERS bool b_RRC_CyclicJob{n_RRC_NumOfCha}:=[FALSE,FALSE,FALSE,FALSE];
    TASK PERS bool b_RRC_CycleTimeRunnig{n_RRC_NumOfCha}:=[FALSE,FALSE,FALSE,FALSE];

    !************************************************
    ! Declaration :     num
    !************************************************
    !
    CONST num n_RRC_NumOfCha:=4;
    !
    CONST num n_RRC_DefaultSocketPortRec{n_RRC_NumOfCha}:=[30101,30102,30103,30104];
    CONST num n_RRC_DefaultSocketPortSen{n_RRC_NumOfCha}:=[30201,30202,30203,30204];
    !
    TASK PERS num n_RRC_ViCustomSocketPortRec{n_RRC_NumOfCha}:=[31101,31102,31103,31104];
    TASK PERS num n_RRC_ViCustomSocketPortSen{n_RRC_NumOfCha}:=[31201,31202,31203,31204];
    !
    TASK PERS num n_RRC_ChaNr:=1;
    TASK PERS num n_RRC_ReadPtrRecBuf{n_RRC_NumOfCha}:=[1,1,1,1];
    TASK PERS num n_RRC_Act_S_ID:=1;
    TASK PERS num n_RRC_CounterFStr{n_RRC_NumOfCha}:=[0,0,0,0];
    TASK PERS num n_RRC_CounterFVal{n_RRC_NumOfCha}:=[0,0,0,0];
    TASK PERS num n_RRC_CyJobStart_S_ID{n_RRC_NumOfCha}:=[1,0,0,0];
    TASK PERS num n_RRC_MinCycleTime{n_RRC_NumOfCha}:=[1,1,1,1];
    TASK PERS num n_RRC_ActCycleTime{n_RRC_NumOfCha}:=[0.364,1,1,1];
    TASK PERS num n_RRC_LastCycleTime{n_RRC_NumOfCha}:=[1.001,1,1,1];
    TASK PERS num n_RRC_ActCycle{n_RRC_NumOfCha}:=[55.002,1,1,1];

    !************************************************
    ! Declaration :     string
    !************************************************
    !
    TASK PERS string st_RRC_ChaTask:="T_ROB1";
    TASK PERS string st_RRC_EvLogMsgHeader:="RRC -- Controller";
    !
    TASK PERS string st_RRC_CyclicJob{n_RRC_NumOfCha}:=["r_RRC_GetJointT","","",""];
    TASK PERS string st_RRC_TPWrite{n_RRC_NumOfCha}:=["E-Level Channel 1 Controller","E-Level Channel 2 Controller","",""];

    !************************************************
    ! Declaration :     jointtarget
    !************************************************
    !
    TASK PERS jointtarget jp_RRC_Act:=[[0,0,0,0,0,0],[9E+09,9E+09,9E+09,9E+09,9E+09,9E+09]];

    !************************************************
    ! Declaration :     robtarget
    !************************************************
    !
    TASK PERS robtarget p_RRC_Act:=[[10270.7,5902.7,955.503],[0.33371,0.672327,0.217398,-0.623981],[1,1,-1,1],[8000,-4200,-2500,0,0,0]];

    !************************************************
    ! Declaration :     string
    !************************************************
    !
    VAR clock ck_RRC_CycleJob{n_RRC_NumOfCha};

    !************************************************
    ! Declaration :     RRC_buffer_msg
    !************************************************
    !
    CONST RRC_buffer_msg bm_RRC_Empty:=[[0,0,0,"",0,0,"",0,0,0,"",0,"",0,"",0,"",0,"",0,"",0,"",0,"",0,0,0,0,0,0,0,0,0,0,0,0,0,0,0,0,0,0,0,0,0,0,0,0,0,0,0,0,0,0,0,0,0,0,0,0,0],FALSE];
    !
    TASK PERS RRC_buffer_msg bm_RRC_ActSenMsgCtrl{n_RRC_NumOfCha}:=[
    [[0,0,0,"",0,0,"",0,0,0,"",0,"",0,"",0,"",0,"",0,"",0,"",0,"",0,0,0,0,0,0,0,0,0,0,0,0,0,0,0,0,0,0,0,0,0,0,0,0,0,0,0,0,0,0,0,0,0,0,0,0,0],FALSE],
    [[0,0,0,"",0,0,"",0,0,0,"",0,"",0,"",0,"",0,"",0,"",0,"",0,"",0,0,0,0,0,0,0,0,0,0,0,0,0,0,0,0,0,0,0,0,0,0,0,0,0,0,0,0,0,0,0,0,0,0,0,0,0],FALSE],
    [[0,0,0,"",0,0,"",0,0,0,"",0,"",0,"",0,"",0,"",0,"",0,"",0,"",0,0,0,0,0,0,0,0,0,0,0,0,0,0,0,0,0,0,0,0,0,0,0,0,0,0,0,0,0,0,0,0,0,0,0,0,0],FALSE],
    [[0,0,0,"",0,0,"",0,0,0,"",0,"",0,"",0,"",0,"",0,"",0,"",0,"",0,0,0,0,0,0,0,0,0,0,0,0,0,0,0,0,0,0,0,0,0,0,0,0,0,0,0,0,0,0,0,0,0,0,0,0,0],FALSE]];

ENDMODULE

--- Backups/vIRB4600-40-2.55-RW11/RAPID/TASK2/SYSMOD/RRC_EULA_Ctrl.sys ---
MODULE RRC_EULA_Ctrl(SYSMODULE)
    !
    !***********************************************************************************************************************
    !
    !                                /########       /##   /##       /##              /######
    !                               | ##_____/      | ##  | ##      | ##             /##__  ##
    !                               | ##            | ##  | ##      | ##            | ##  \ ##
    !                               | #####         | ##  | ##      | ##            | ########
    !                               | ##__/         | ##  | ##      | ##            | ##__  ##
    !                               | ##            | ##  | ##      | ##            | ##  | ##
    !                               | ########      |  ######/      | ########      | ##  | ##
    !                               |________/       \______/       |________/      |__/  |__/
    !
    !***********************************************************************************************************************
    !
    !
    ! THIS EULA IS INTENDED ONLY FOR PRIVATE, INDIVIDUAL AND NON-COMMERCIAL USE OR FOR NON-COMMERCIAL ACADEMIC USE.
    ! IF YOU INTEND TO USE THE SOFTWARE FOR DIFFERENT PURPOSES (e.g. COMMERCIAL) PLEASE CONTACT: rrc@arch.ethz.ch
    ! This End-User License Agreement ("EULA") is a legal agreement between you ("You") (either an individual or a person
    ! acting on behalf of a legal entity) and ETH Zurich, Raemistrasse 101, 8092 Zurich (Switzerland) ("ETH Zurich") for
    ! the "Rapid Robot Communication Server for ABB Robots" which includes computer software and associated media, and may
    ! include "online" or electronic documentation ("SOFTWARE"). The SOFTWARE enables the dynamic communication of a robot
    ! system. Dynamic communication means that changing contents can be transferred into production commands without the
    ! need for individual programming of the production commands for each design. Furthermore, the SOFTWARE enables feedback
    ! from previous production commands in order to adapt the current product (e.g. to react to process tolerances). The
    ! SOFTWARE is installed on the robot control and any client with the appropriate interface (e.g. COMPAS_RRC) can connect
    ! to this server. The SOFTWARE is protected by copyright laws. The SOFTWARE is hereby licensed, not sold. In order to
    ! use the SOFTWARE, You must indicate agreement with the following terms and conditions by signing this EULA. If You are
    ! accepting the terms for use in this EULA on behalf of an organization, You herewith represent that You have the
    ! authority to enter into this EULA.
    !
    !
    ! 1 LICENSE GRANT
    !
    ! (i) ETH Zurich hereby grants to You a free-of-charge, single, non-exclusive, world-wide, non-transferable,
    ! non-sublicensable right to install, execute and display the encrypted part of the SOFTWARE and to develop, modify,
    ! adapt and/or create derivative works, install, execute and display the human readable part of the SOFTWARE on a single
    ! device running a validly licensed copy of the operating system for which the SOFTWARE was designed. Such rights are
    ! granted for the sole purpose for (i) private and non-commercial use or for (ii) non-commercial academic use. You are
    ! NOT allowed to use the SOFTWARE for any commercial purposes.
    !
    ! (ii) With respect to electronic documents included with the SOFTWARE, you may make an unlimited number of copies
    ! (either in hardcopy or electronic form), provided that such copies shall be used only for internal purposes and are
    ! not republished or distributed to any third party.
    !
    !
    ! 2 USE OF RESULTS GENERATED BY THE SOFTWARE
    !
    ! You are only allowed to use the content generated by the SOFTWARE ("SOFTWARE RESULTS") for private, individual and
    ! non-commercial purposes or for non-commercial academic purposes. Any use of the SOFTWARE RESULTS outside these purposes
    ! is strictly forbidden. Note that any attribution (e.g. ETH Zurich logo or the name of data provider) on the SOFTWARE
    ! RESULTS must be retained. You are not allowed to alter, cancel or fade, after a few seconds, such attribution.
    !
    !
    ! 3 DURATION OF LICENSE AND TERMINATION
    !
    ! This EULA enters into effect on the date of acceptance of this EULA by You. This EULA,
    ! (i) may be terminated by ETH Zurich at any time for any reason;
    !
    ! (ii) will terminate automatically without notice from ETH Zurich if (a) You fail to comply with any term(s) of this
    ! EULA or (b) You refuse, after the notification in accordance with clause 10 (i), to accept the new EULA term and
    ! conditions provided by ETH Zurich;
    !
    ! (iii) is terminated as soon as You cease to use the SOFTWARE and destroy all copies, full or partial, of the SOFTWARE;
    ! Upon termination pursuant to (i) and (ii), you must cease all use of the SOFTWARE and destroy all copies, full or
    ! partial, of the SOFTWARE.
    !
    !
    ! 4 OBLIGATIONS OF YOU
    !
    ! (i) You may not remove or alter any copyright notices on any and all copies of the SOFTWARE.
    !
    ! (ii) You may not distribute or assign the SOFTWARE or any copy thereof to third parties. You may not rent, lease,
    ! sell, lend, transfer, redistribute, or sublicense the SOFTWARE to any third party.
    !
    ! (iii) You may not reverse engineer, decompile or disassemble the SOFTWARE, except and only to the extent that such
    ! activity is expressly permitted by applicable law despite this limitation.
    !
    ! (iv) You may not reproduce and copy the SOFTWARE, except and only to the extent that such activity is expressly
    ! permitted by applicable law despite this limitation.
    !
    ! (v) You must comply with all applicable laws.
    !
    !
    ! 5 OWNERSHIP
    !
    ! Except as expressly licensed to You in this EULA, ETH Zurich and its licensors retains all right, title, and interest
    ! in and to the SOFTWARE. All title and copyrights in and to the SOFTWARE (including but not limited to any images,
    ! photographs, animations, video, audio, music, text, and "applets" incorporated into the SOFTWARE), the accompanying
    ! materials, and any copies of the SOFTWARE are owned by ETH Zurich and its licensors. The SOFTWARE is protected by
    ! copyright laws. Therefore, You must treat the SOFTWARE like any other copyrighted material. All rights not expressly
    ! granted are reserved by ETH Zurich.
    !
    !
    ! 6 MAINTENANCE, SUPPORT, UPGRADES OR NEW RELEASES
    !
    ! ETH Zurich has no obligation to provide maintenance, support, upgrades, new releases, enhancements or modifications
    ! and disclaims all costs associated with service, repair or correction of the SOFTWARE. If any supplemental software
    ! code is provided by ETH Zurich to You this supplemental software code shall be considered part of the SOFTWARE and is
    ! subject to the terms and conditions of this EULA. It is expressly acknowledged by You that no rights to receive
    ! upgrades may be derived from this EULA.
    !
    !
    ! 7 NO WARRANTY
    !
    ! YOU EXPRESSLY ACKNOWLEDGE AND AGREE THAT USE OF THE SOFTWARE IS AT YOUR SOLE RISK AND THAT THE ENTIRE RISK AS TO
    ! SATISFACTORY QUALITY, PERFORMANCE, ACCURACY, AND EFFORT IS WITH YOU. TO THE MAXIMUM EXTENT PERMITTED BY APPLICABLE LAW,
    ! THE SOFTWARE AND ANY SERVICES PERFORMED OR PROVIDED BY THE SOFTWARE ARE PROVIDED "AS IS" AND "AS AVAILABLE",
    ! WITH ALL FAULTS AND WITHOUT WARRANTY OF ANY KIND, AND ETH ZURICH HEREBY DISCLAIMS ALL WARRANTIES AND CONDITIONS
    ! WITH RESPECT TO THE SOFTWARE AND ANY SERVICES, EITHER EXPRESS, IMPLIED, OR STATUTORY, INCLUDING, BUT NOT LIMITED TO,
    ! THE IMPLIED WARRANTIES AND/OR CONDITIONS OF MERCHANTABILITY, OF SATISFACTORY QUALITY, OF FITNESS FOR A PARTICULAR
    ! PURPOSE, OF ACCURACY, OF QUIET ENJOYMENT, AND OF NON-INFRINGEMENT OF THIRD-PARTY RIGHTS. ETH ZURICH DOES NOT WARRANT
    ! AGAINST INTERFERENCE WITH YOUR ENJOYMENT OF THE SOFTWARE, THAT THE FUNCTIONS CONTAINED IN OR SERVICES PERFORMED OR
    ! PROVIDED BY THE SOFTWARE WILL MEET YOUR REQUIREMENTS, THAT THE OPERATION OF THE SOFTWARE OR SERVICES WILL BE
    ! UNINTERRUPTED OR ERROR-FREE, OR THAT DEFECTS IN THE SOFTWARE OR SERVICES WILL BE CORRECTED. NO ORAL OR WRITTEN
    ! INFORMATION OR ADVICE GIVEN BY ETH ZURICH OR ITS AUTHORIZED REPRESENTATIVE SHALL CREATE A WARRANTY. SHOULD THE
    ! SOFTWARE OR SERVICES PROVE DEFECTIVE, YOU ASSUME THE ENTIRE COST OF ALL NECESSARY SERVICING, REPAIR, OR CORRECTION.
    ! SOME JURISDICTIONS DO NOT ALLOW THE EXCLUSION OF IMPLIED WARRANTIES OR LIMITATIONS ON APPLICABLE STATUTORY RIGHTS
    ! OF A CONSUMER, SO THE ABOVE EXCLUSION AND LIMITATIONS MAY NOT APPLY TO YOU.
    !
    !
    ! 8 LIABILITY
    !
    ! In no event shall ETH Zurich be liable for any damages (including, without limitation, lost profits, business
    ! interruption, or lost information) arising from the use of or inability to use the SOFTWARE through You.
    ! In no event will ETH Zurich be liable for loss of data or for indirect, special, incidental, consequential
    ! (including lost profit), or other damages based in contract, tort or otherwise. The above limitation of liability
    ! shall not be construed to amend or limit any Party's statutory liability.
    !
    !
    ! 9 GENERAL PROVISIONS
    !
    ! (i) ETH Zurich reserves the right to change the terms and conditions of this EULA at any point in time. In such event,
    ! ETH Zurich will notify You in due time of the changes to the terms of the EULA.
    !
    ! (ii) Rights and duties derived from this EULA shall not be transferred to third parties without the written
    ! acceptance of the ETH Zurich.
    !
    ! (iii) You shall not infer from this EULA any other rights, including licenses, than those that are explicitly stated herein.
    !
    ! (iv) This EULA shall exclusively be governed by and interpreted in accordance with the laws of Switzerland,
    ! without reference to its conflict of laws principles. The exclusive place of jurisdiction is Zurich (Switzerland).
    !
    !
    ! 10 AKNOWLEDGMENT
    !
    ! You acknowledge that you have read this EULA, understand it, and had an opportunity to seek independent legal advice prior
    ! to agreeing to it. In consideration of ETH Zurich agreeing to provide the SOFTWARE, You agree to be bound by the terms and
    ! conditions of this EULA. You further agree that it is the complete and exclusive statement of the agreement between you and
    ! ETH Zurich, which supersedes any proposal or prior agreement, oral or written, and any other communication between you and
    ! ETH Zurich relating to the subject of this EULA.
    !
ENDMODULE

--- Backups/vIRB4600-40-2.55-RW11/RAPID/TASK2/SYSMOD/RRC_Helper_Ctrl.sys ---
MODULE RRC_Helper_Ctrl(SYSMODULE)
    !***********************************************************************************
    !
    ! ETH Zurich / Robotic Fabrication Lab
    ! HIB C 13 / Stefano-Franscini-Platz 1
    ! CH-8093 Zurich
    !
    !***********************************************************************************
    !
    ! PROJECT     :  RRC - Rapid Robot Communication
    !
    ! FUNCTION    :  Helper routines for project
    !
    ! AUTHOR      :  Philippe Fleischmann
    !
    ! EMAIL       :  rrc@arch.ethz.ch
    !
    ! HISTORY     :  2019.02.22
    !
    ! Copyright   :  ETH Zurich (CH) 2019
    !                - Philippe Fleischmann
    !                - Michael Lyrenmann
    !                - Gonzalo Casas
    !
    ! License     :  This code base is governed by an EULA (End-User License Agreement)
    !                which you have received together with the software.
    !                You are not allowed to use the software on a real robots
    !                without a signed EULA.
    !
    !                A copy of the EULA content is in the controller task (T_CTRL).
    !
    !***********************************************************************************


ENDMODULE

--- Backups/vIRB4600-40-2.55-RW11/RAPID/TASK2/SYSMOD/RRC_UserInteraction.sys ---
MODULE RRC_UserInteraction(SYSMODULE,NOSTEPIN)
    !***********************************************************************************
    !
    ! ETH Zurich / Robotic Fabrication Lab
    ! HIB C 13 / Stefano-Franscini-Platz 1
    ! CH-8093 Zurich
    !
    !***********************************************************************************
    !
    ! PROJECT     :  RRC - Rapid Robot Communication
    !
    ! FUNCTION    :  General Utilities Library
    !
    ! AUTHOR      :  Philippe Fleischmann
    !
    ! EMAIL       :  rrc@arch.ethz.ch
    !
    ! HISTORY     :  2019.02.22
    !
    ! Copyright   :  ETH Zurich (CH) 2019
    !                - Philippe Fleischmann
    !                - Michael Lyrenmann
    !                - Gonzalo Casas
    !
    ! License     :  This code base is governed by an EULA (End-User License Agreement)
    !                which you have received together with the software.
    !                You are not allowed to use the software on a real robots
    !                without a signed EULA.
    !
    !                A copy of the EULA content is in the controller task (T_CTRL).
    !
    !***********************************************************************************

    !************************************************
    ! Function    :     Teach Pendant (old FelxPendant) Message
    ! Programmer  :     Philippe Fleischmann
    ! Date        :     2019.02.22
    !***************** ETH Zurich *******************
    !
    PROC r_RRC_TPMsg(string stMsg)
        !
        ! Clear Msg Panel
        TPErase;
        !
        ! Msg for user
        TPWrite stMsg;
        !
        ! Time to read the Msg
        WaitTime n_RRC_TimeTPMsg;
        RETURN ;
    ERROR
        ! Placeholder for Error Code...
    ENDPROC

    !************************************************
    ! Function    :     Teach Pendant (old FelxPendant) Error Message
    ! Programmer  :     Philippe Fleischmann
    ! Date        :     2019.02.22
    !***************** ETH Zurich *******************
    !
    PROC r_RRC_TPErrMsg(num nErrno\switch StopTask\switch StopAllTasks)
        !
        ! Clear Msg Panel
        TPErase;
        !
        ! Write error number
        TPWrite "ERRNO = "\Num:=nErrno;
        !
        ! Stop task
        IF Present(StopTask) Stop;
        !
        ! Stop all normal tasks
        IF Present(StopAllTasks) Stop\AllMoveTasks;
        RETURN ;
    ERROR
        ! Placeholder for Error Code...
    ENDPROC

    !************************************************
    ! Function    :     Event Log Message
    ! Programmer  :     Philippe Fleischmann
    ! Date        :     2019.02.22
    !***************** ETH Zurich *******************
    !
    PROC r_RRC_EvLogMsg(string stHeader,string stMsg)
        !
        ! Msg for user
        ErrWrite\I,stHeader+" "+stMsg,"rLogMsg";
        RETURN ;
    ERROR
        ! Placeholder for Error Code...
    ENDPROC

    !************************************************
    ! Function    :     User interface message
    ! Programmer  :     Philippe Fleischmann
    ! Date        :     2019.02.22
    !***************** ETH Zurich *******************
    !
    FUNC string f_RRC_UIMsg(string stMsgHeader,string stMsgL1,\string stMsgL2,\string stMsgL3,\string stMsgL4,\string stMsgL5,string stBtn1\string stBtn2\string stBtn3\string stBtn4\string stBtn5,icondata icIcon)
        VAR num nAnswer;
        VAR string stMsg{5};
        VAR string stBtn{5};
        VAR string stAnswer;
        !
        ! Initialize variables
        stMsg:=["","","","",""];
        stBtn:=["","","","",""];
        !
        ! Load meassge
        stMsg{1}:=stMsgL1;
        IF Present(stMsgL2) stMsg{2}:=stMsgL2;
        IF Present(stMsgL3) stMsg{3}:=stMsgL3;
        IF Present(stMsgL4) stMsg{4}:=stMsgL4;
        IF Present(stMsgL5) stMsg{5}:=stMsgL5;
        !
        ! Load buttons
        stBtn{1}:=stBtn1;
        IF Present(stBtn2) stBtn{2}:=stBtn2;
        IF Present(stBtn3) stBtn{3}:=stBtn3;
        IF Present(stBtn4) stBtn{4}:=stBtn4;
        IF Present(stBtn5) stBtn{5}:=stBtn5;
        !
        ! Msg for user
        nAnswer:=UIMessageBox(
            \Header:=stMsgHeader
            \MsgArray:=stMsg
            \BtnArray:=stBtn
            \Icon:=icIcon);
        !
        ! handle user answer
        IF nAnswer=1 stAnswer:=stBtn{1};
        IF nAnswer=2 stAnswer:=stBtn{2};
        IF nAnswer=3 stAnswer:=stBtn{3};
        IF nAnswer=4 stAnswer:=stBtn{4};
        IF nAnswer=5 stAnswer:=stBtn{5};
        !
        ! Return user answer as string
        RETURN stAnswer;
    ERROR
        ! Placeholder for Error Code...
    ENDFUNC

    !************************************************
    ! Function    :     User interface numerical entry
    ! Programmer  :     Philippe Fleischmann
    ! Date        :     2019.02.22
    !***************** ETH Zurich *******************
    !
    FUNC num f_RRC_UINumEntry(string stMsgHeader,string stMsgL1,\string stMsgL2,\string stMsgL3,\string stMsgL4,\string stMsgL5,num nMin,num nMax,\num nDefault,icondata icIcon)
        VAR string stMsg{5};
        VAR num nAnswer;
        VAR num nInitValue;
        !
        ! Initialize variables
        stMsg:=["","","","",""];
        nInitValue:=nMin;
        !
        ! Load meassge
        stMsg{1}:=stMsgL1;
        IF Present(stMsgL2) stMsg{2}:=stMsgL2;
        IF Present(stMsgL3) stMsg{3}:=stMsgL3;
        IF Present(stMsgL4) stMsg{4}:=stMsgL4;
        IF Present(stMsgL5) stMsg{5}:=stMsgL5;
        !
        ! Use default value when present
        IF Present(nDefault) nInitValue:=nDefault;
        !
        ! Msg for user
        nAnswer:=Round(UINumEntry(
            \Header:=stMsgHeader
            \MsgArray:=stMsg
            \Icon:=icIcon
            \InitValue:=nInitValue
            \MinValue:=nMin
            \MaxValue:=nMax)\Dec:=1);
        !
        ! Return user answer as string
        RETURN nAnswer;
    ERROR
        ! Placeholder for Error Code...
    ENDFUNC


ENDMODULE

